// TwinCAT 3 PLC project MAIN
// ProgramVersion: 3.1.0.5
// libraries:
//   Tc2_ModbusRTU, * (Beckhoff Automation GmbH)
//   Tc2_Standard, * (Beckhoff Automation GmbH)
//   Tc2_System, * (Beckhoff Automation GmbH)
//   Tc2_Utilities, * (Beckhoff Automation GmbH)
//   Tc2_XmlDataSrv, * (Beckhoff Automation GmbH)
//   Tc3_Interfaces, * (Beckhoff Automation GmbH)
//   Tc3_Module, * (Beckhoff Automation GmbH)
//   VisuDialogs, * (System)
// project tree:
//   DUTs/ RESET_STATE.TcDUT, ST_DisplayPositions.TcDUT, ST_SavedStructure.TcDUT, ST_SavedPositions.TcDUT, SYSTEM_STATE.TcDUT
//   / GlobalTextList.TcGTLO, PlcTask.TcTTO, Visualization Manager.TcVMO (not stored), VISU_TASK.TcTTO
//   GVLs/ GV_HMI.TcGVL, GV_LIFT.TcGVL, GV_MODBUS.TcGVL
//   POUs/ HMI.TcPOU, IO_SWITCHBOARD.TcPOU, MAIN.TcPOU, MOVE_TO_POSITION.TcPOU, SYSTEM_RESET.TcPOU, XML.TcPOU
//   POUs/HMI/ HMI_Crush_Indicator.TcPOU, HMI_Door_Toggle.TcPOU, HMI_Down_Arrow_Indicator.TcPOU, HMI_Hard_Limits.TcPOU, HMI_System_Indicator.TcPOU, HMI_Ultimate_Limit.TcPOU, HMI_Up_Arrow_Indicator.TcPOU
//   POUs/Pendant Screen/ DoorFaults.TcPOU, DownLimit.TcPOU, EStop.TcPOU, JogLift.TcPOU, MoveToPosition.TcPOU, ReadWriteScreen.TcPOU, SelectSpike.TcPOU, SwitchScreens.TcPOU, UpLimit.TcPOU
//   POUs/Pendant Screen/Functions/ Execute_Write_Screen.TcPOU, Fill_Row_Four.TcPOU, Fill_Row_Three.TcPOU, Fill_Row_Two.TcPOU, Get_Valid_Indexs.TcPOU, Position_To_Row_Array.TcPOU, Spike_To_Half_Row_Array.TcPOU, Spike_To_Row_Array.TcPOU
//   VISUs/ MAIN_DASHBOARD.TcVIS, SAFETY_PANEL.TcVIS, TARGET_PANEL.TcVIS
// real-time tasks:
//   TASK PlcTask: cycle T#15ms, priority 20, ADS port 350
//   TASK VISU_TASK: cycle T#20ms, priority 30, ADS port 351
// I/O:
//   DEVICE Device 1 (EtherCAT), AmsNetId 5.31.29.63.2.1
//     Term 1 (EK1200) [EK1200-5000 EtherCAT Power supply (2A E-Bus)]
//       Term 2 (EL1904) [EL1904, 4 Ch. Safety Input 24V, TwinSAFE]
//         modules: Module 1 (FSOES)
//       Term 3 (EL1859) [EL1859 8Ch. Dig. Input 24V, 3ms, 8Ch. Dig. Output 24V, 0.5A]
//       Term 4 (EK1110) [EK1110 EtherCAT extension]
//     Term 5 (EK1914) [EK1914, 2 Ch. Safety Input/Output 24V,  TwinSAFE]
//       modules: Module 1 (FSOE), Module 2 (DIO)
//       Term 6 (EL1904) [EL1904, 4 Ch. Safety Input 24V, TwinSAFE]
//         modules: Module 1 (FSOES)
//       Term 7 (EL6021) [EL6021 Interface (RS422/485)]
//       Term 15 (EL9011) [EL9011 End Terminal]
//     Term 8 (EK1100) [EK1100 EtherCAT Coupler (2A E-Bus)]
//       Term 9 (EL6900) [EL6900, TwinSAFE PLC]
//       Term 10 (EL1904) [EL1904, 4 Ch. Safety Input 24V, TwinSAFE]
//         modules: Module 1 (FSOES)
//       Term 11 (EL1904) [EL1904, 4 Ch. Safety Input 24V, TwinSAFE]
//         modules: Module 1 (FSOES)
//       Term 12 (EL1904) [EL1904, 4 Ch. Safety Input 24V, TwinSAFE]
//         modules: Module 1 (FSOES)
//       Term 13 (EL1904) [EL1904, 4 Ch. Safety Input 24V, TwinSAFE]
//         modules: Module 1 (FSOES)
//       Term 16 (EL9011) [EL9011 End Terminal]
//     Box 14 (SICK AFS60A ST, 18-Bit) [AFS60A_ST 18-Bit]
// variable links:
//   Device 1 (EtherCAT) <-> Device 1 (EtherCAT)/Term 1 (EK1200)/Term 2 (EL1904)
//     Term 8 (EK1100)/ConnectionOutputs/Message_86 RxPDO <-> Module 1 (FSOES)/TxPDO/FSOE
//     Term 8 (EK1100)/Term 9 (EL6900)/ConnectionOutputs/Message_86 RxPDO <-> Module 1 (FSOES)/TxPDO/FSOE
//   Device 1 (EtherCAT) <-> Device 1 (EtherCAT)/Term 5 (EK1914)
//     Term 8 (EK1100)/Term 9 (EL6900)/ConnectionInputs/Message_87 TxPDO <-> Module 1 (FSOE)/Outputs/FSOE
//   Device 1 (EtherCAT) <-> Device 1 (EtherCAT)/Term 5 (EK1914)/Term 6 (EL1904)
//     Term 8 (EK1100)/Term 9 (EL6900)/ConnectionOutputs/Message_88 RxPDO <-> Module 1 (FSOES)/TxPDO/FSOE
//   Device 1 (EtherCAT) <-> Device 1 (EtherCAT)/Term 8 (EK1100)
//     Term 5 (EK1914)/Term 6 (EL1904)/Module 1 (FSOES)/TxPDO/FSOE <-> ConnectionOutputs/Message_88 RxPDO
//     Term 8 (EK1100)/Term 11 (EL1904)/Module 1 (FSOES)/TxPDO/FSOE <-> ConnectionOutputs/Message_90 RxPDO
//     Term 8 (EK1100)/Term 13 (EL1904)/Module 1 (FSOES)/TxPDO/FSOE <-> ConnectionOutputs/Message_92 RxPDO
//   Device 1 (EtherCAT) <-> Device 1 (EtherCAT)/Term 8 (EK1100)/Term 10 (EL1904)
//     Term 8 (EK1100)/ConnectionOutputs/Message_89 RxPDO <-> Module 1 (FSOES)/TxPDO/FSOE
//     Term 8 (EK1100)/Term 9 (EL6900)/ConnectionInputs/Message_89 TxPDO <-> Module 1 (FSOES)/RxPDO/FSOE
//   Device 1 (EtherCAT) <-> Device 1 (EtherCAT)/Term 8 (EK1100)/Term 11 (EL1904)
//     Term 8 (EK1100)/Term 9 (EL6900)/ConnectionOutputs/Message_90 RxPDO <-> Module 1 (FSOES)/TxPDO/FSOE
//   Device 1 (EtherCAT) <-> Device 1 (EtherCAT)/Term 8 (EK1100)/Term 12 (EL1904)
//     Term 8 (EK1100)/ConnectionOutputs/Message_91 RxPDO <-> Module 1 (FSOES)/TxPDO/FSOE
//     Term 8 (EK1100)/Term 9 (EL6900)/ConnectionInputs/Message_91 TxPDO <-> Module 1 (FSOES)/RxPDO/FSOE
//   Device 1 (EtherCAT) <-> Device 1 (EtherCAT)/Term 8 (EK1100)/Term 13 (EL1904)
//     Term 8 (EK1100)/Term 9 (EL6900)/ConnectionOutputs/Message_92 RxPDO <-> Module 1 (FSOES)/TxPDO/FSOE
//   Device 1 (EtherCAT) <-> Device 1 (EtherCAT)/Term 8 (EK1100)/Term 9 (EL6900)
//     Term 1 (EK1200)/Term 2 (EL1904)/Module 1 (FSOES)/RxPDO/FSOE <-> ConnectionInputs/Message_86 TxPDO
//     Term 5 (EK1914)/Term 6 (EL1904)/Module 1 (FSOES)/RxPDO/FSOE <-> ConnectionInputs/Message_88 TxPDO
//     Term 8 (EK1100)/Term 11 (EL1904)/Module 1 (FSOES)/RxPDO/FSOE <-> ConnectionInputs/Message_90 TxPDO
//     Term 8 (EK1100)/Term 13 (EL1904)/Module 1 (FSOES)/RxPDO/FSOE <-> ConnectionInputs/Message_92 TxPDO
//     Term 5 (EK1914)/Module 1 (FSOE)/Inputs/FSOE <-> ConnectionOutputs/Message_87 RxPDO
//     Term 8 (EK1100)/Term 10 (EL1904)/Module 1 (FSOES)/TxPDO/FSOE <-> ConnectionOutputs/Message_89 RxPDO
//     Term 8 (EK1100)/Term 12 (EL1904)/Module 1 (FSOES)/TxPDO/FSOE <-> ConnectionOutputs/Message_91 RxPDO
//   MAIN/MAIN Instance <-> Device 1 (EtherCAT)/Box 14 (SICK AFS60A ST, 18-Bit)
//     PlcTask Inputs/MOVE_TO_POSITION.currentRawPosition <-> TxPDO-1/Position Value
//   MAIN/MAIN Instance <-> Device 1 (EtherCAT)/Term 1 (EK1200)/Term 3 (EL1859)
//     PlcTask Inputs/GV_LIFT.LIMIT_OVERRIDE_BUTTON_IN <-> Channel 1/Input
//     PlcTask Inputs/IO_SWITCHBOARD.CONSOLE_DOWN_BUTTON_IN <-> Channel 3/Input
//     PlcTask Inputs/IO_SWITCHBOARD.CONSOLE_RESET_BUTTON_IN <-> Channel 5/Input
//     PlcTask Inputs/IO_SWITCHBOARD.CONSOLE_RUN_BUTTON_IN <-> Channel 4/Input
//     PlcTask Inputs/IO_SWITCHBOARD.CONSOLE_UP_BUTTON_IN <-> Channel 2/Input
//   MAIN/MAIN Instance <-> Device 1 (EtherCAT)/Term 5 (EK1914)
//     PlcTask Inputs/IO_SWITCHBOARD.REMOTE_DOWN_BUTTON_IN <-> Module 2 (DIO)/DIO Inputs/Input 1
//     PlcTask Inputs/IO_SWITCHBOARD.REMOTE_RESET_BUTTON_IN <-> Module 2 (DIO)/DIO Inputs/Input 0
//     PlcTask Inputs/IO_SWITCHBOARD.REMOTE_RUN_BUTTON_IN <-> Module 2 (DIO)/DIO Inputs/Input 3
//     PlcTask Inputs/IO_SWITCHBOARD.REMOTE_UP_BUTTON_IN <-> Module 2 (DIO)/DIO Inputs/Input 2
//   MAIN/MAIN Instance <-> Device 1 (EtherCAT)/Term 5 (EK1914)/Term 7 (EL6021)
//     PlcTask Inputs/GV_MODBUS.screen.InData/D[{0..21}] <-> COM TxPDO-Map Inputs/Data In {0..21}  (22 links)
//     PlcTask Inputs/GV_MODBUS.screen.InData/Status <-> COM TxPDO-Map Inputs/Status
//     PlcTask Outputs/GV_MODBUS.screen.OutData/Ctrl <-> COM RxPDO-Map Outputs/Ctrl
//     PlcTask Outputs/GV_MODBUS.screen.OutData/D[{0..21}] <-> COM RxPDO-Map Outputs/Data Out {0..21}  (22 links)
//   MAIN/MAIN Instance <-> Device 1 (EtherCAT)/Term 8 (EK1100)/Term 9 (EL6900)
//     PlcTask Inputs/GV_LIFT.CONSOLE_ESTOP_INDICATOR_IN <-> StandardInputs/Standard Out Var 68
//     PlcTask Inputs/GV_LIFT.CRUSH_PROTECTION_INDICATOR_IN <-> StandardInputs/Standard Out Var 60
//     PlcTask Inputs/GV_LIFT.DOOR_{1..4}_INDICATOR_IN <-> StandardInputs/Standard Out Var {56..59}  (4 links)
//     PlcTask Inputs/GV_LIFT.DOOR_{1..4}_INDICATOR_LATCH_IN <-> StandardInputs/Standard Out Var {72..75}  (4 links)
//     PlcTask Inputs/GV_LIFT.DOWNSTAGE_ESTOP_INDICATOR_IN <-> StandardInputs/Standard Out Var 70
//     PlcTask Inputs/GV_LIFT.DOWN_INDICATOR_IN <-> StandardInputs/Standard Out Var 63
//     PlcTask Inputs/GV_LIFT.DOWN_LIMIT_INDICATOR_IN <-> StandardInputs/Standard Out Var 65
//     PlcTask Inputs/GV_LIFT.DOWN_LIMIT_INDICATOR_LATCH_IN <-> StandardInputs/Standard Out Var 77
//     PlcTask Inputs/GV_LIFT.ESTOP_INDICATOR_IN <-> StandardInputs/Standard Out Var 61
//     PlcTask Inputs/GV_LIFT.FAULT_INDICATOR_IN <-> StandardInputs/Standard Out Var 62
//     PlcTask Inputs/GV_LIFT.PIT_ESTOP_INDICATOR_IN <-> StandardInputs/Standard Out Var 67
//     PlcTask Inputs/GV_LIFT.PUMP_ESTOP_INDICATOR_IN <-> StandardInputs/Standard Out Var 69
//     PlcTask Inputs/GV_LIFT.REMOTE_ESTOP_INDICATOR_IN <-> StandardInputs/Standard Out Var 71
//     PlcTask Inputs/GV_LIFT.ULTIMATE_LIMIT_INDICATOR_IN <-> StandardInputs/Standard Out Var 66
//     PlcTask Inputs/GV_LIFT.ULTIMATE_LIMIT_INDICATOR_LATCH_IN <-> StandardInputs/Standard Out Var 78
//     PlcTask Inputs/GV_LIFT.UPSTAGE_ESTOP_INDICATOR_IN <-> StandardInputs/Standard Out Var 55
//     PlcTask Inputs/GV_LIFT.UP_INDICATOR_IN <-> StandardInputs/Standard Out Var 54
//     PlcTask Inputs/GV_LIFT.UP_LIMIT_INDICATOR_IN <-> StandardInputs/Standard Out Var 64
//     PlcTask Inputs/GV_LIFT.UP_LIMIT_INDICATOR_LATCH_IN <-> StandardInputs/Standard Out Var 76
//     PlcTask Outputs/GV_LIFT.DOWN_BUTTON_OUT <-> StandardOutputs/Standard In Var 53
//     PlcTask Outputs/GV_LIFT.UP_BUTTON_OUT <-> StandardOutputs/Standard In Var 52
//     PlcTask Outputs/SYSTEM_RESET.ERROR_ACKNOWLEDGEMENT_BUTTON_OUT <-> StandardOutputs/Standard In Var 1
//     PlcTask Outputs/SYSTEM_RESET.ESTOP_RESTART_BUTTON_OUT <-> StandardOutputs/Standard In Var 10

CONFIGURATION MAIN
    RESOURCE PLC ON TwinCAT3
        TASK PlcTask(INTERVAL := T#20ms, PRIORITY := 20);
        TASK VISU_TASK(INTERVAL := T#30ms, PRIORITY := 30);
        PROGRAM MAIN WITH PlcTask : MAIN;
        PROGRAM VisuElems_Visu_Prg WITH VISU_TASK : VisuElems.Visu_Prg;
    END_RESOURCE
END_CONFIGURATION

// ---- DUTs/RESET_STATE.TcDUT
{attribute 'qualified_only'}
{attribute 'strict'}
TYPE RESET_STATE :
(
	IDLE,
	ERRACK_ON,
	ERRACK_OFF,
	IDLE2,
	ESTOP_RESET_ON,
	COMPLETE
);
END_TYPE

// ---- DUTs/ST_DisplayPositions.TcDUT
TYPE ST_DisplayPositions :
STRUCT
	target		:	STRING;
	description	:	STRING;
END_STRUCT
END_TYPE

// ---- DUTs/ST_SavedStructure.TcDUT
TYPE ST_SavedStructure :
STRUCT
	rStagePosition 	:	REAL;
	UpSoftLim		:	REAL;
	DownSoftLim		:	REAL;
	Counter			:	INT;
	SavedPos		:	ARRAY [1..25] OF ST_SavedPositions;
END_STRUCT
END_TYPE

// ---- DUTs/ST_SavedPositions.TcDUT
TYPE ST_SavedPositions :
STRUCT
	target		:	REAL;
	description	:	STRING;
	targetclear	:	BOOL:=FALSE;
END_STRUCT
END_TYPE

// ---- DUTs/SYSTEM_STATE.TcDUT
{attribute 'qualified_only'}
{attribute 'strict'}
TYPE SYSTEM_STATE :
(
	SYSTEM_READY,
	CONSOLE_CONTROL,
	REMOTE_CONTROL
);
END_TYPE

// ---- GVLs/GV_HMI.TcGVL
{attribute 'qualified_only'}
VAR_GLOBAL CONSTANT
	iMaxTargets		:	INT:=25;
	iMaxButtons		:	INT:=20;

END_VAR

VAR_GLOBAL
	ColorToggle		  :	ARRAY [1..20] OF BOOL;

	CurrentPos		:	REAL:=100;
	updatedPos  	:   REAL;
	RowSelect		:	INT:=1;
	ColumnSelect	:	INT:=1;
	RowSelected		:	INT:= RowSelect;


	dwRed				: DWORD:= 16#FFFF0000;
	dwGreen				: DWORD:= 16#FF008040;
	dwYellow			: DWORD:= 16#FFFFFF00;
	dwGrey				: DWORD:= 16#FFBEBEBE;
	
END_VAR

// ---- GVLs/GV_LIFT.TcGVL
{attribute 'qualified_only'}

(*
Signal Flow:

 Physical/HMI Button ---> *_BUTTON_IN ---> *_BUTTON_OUT ---> *_SAFETY_IN ---> *_SAFETY_OUT ---> *_INDICATOR_IN ---> *_INDICATOR_OUT
|------PHYSICAL-----|    |--------IO_SWITCHBOARD-------|    |-------SAFETY PROJECT--------|    |-----------IO_SWITCHBOARD-----------|

This convolution is based on the alias device scheme in the safety project. Recall that an input alias in the safety project must be 
mapped to a PLC/Physical output, and vice versa. The IO_SWITCHBOARD handles signal passthroughs and negotiations between operator
stations. Variables in this GVL should reflect the accurate state of signals to/from the machine. As such, the UP/DOWN/RUN buttons
should reference the appropriate local variables in IO_SWITCHBOARD, which will route signals to the UP/DOWN/RUN_BUTTON_OUT outputs in
this GVL.
*)
VAR_GLOBAL
	REMOTE_ACTIVE_INDICATOR_OUT AT %Q* : BOOL;
	CONSOLE_ACTIVE_INDICATOR_OUT AT %Q* : BOOL;
	
	SYSTEM_RESET_BUTTON_IN AT %I*: BOOL;
	
	//UP_BUTTON_IN AT %I* : BOOL;
	UP_BUTTON_OUT AT %Q* : BOOL;
	
	UP_INDICATOR_IN AT %I* : BOOL;
	UP_INDICATOR_OUT AT %Q* : BOOL;
	
	//DOWN_BUTTON_IN AT %I* : BOOL;
	DOWN_BUTTON_OUT AT %Q* : BOOL;
	
	DOWN_INDICATOR_IN AT %I* : BOOL;
	DOWN_INDICATOR_OUT AT %Q* : BOOL;

	//RUN_BUTTON_IN AT %I* : BOOL;
	RUN_BUTTON_OUT AT %Q* : BOOL;
	
	DOOR_1_INDICATOR_IN AT %I* : BOOL;
	DOOR_1_INDICATOR_OUT AT %Q* : BOOL;
	
	DOOR_1_INDICATOR_LATCH_IN AT %I* : BOOL;
	DOOR_1_INDICATOR_LATCH_OUT AT %Q* : BOOL;
	
	DOOR_2_INDICATOR_IN AT %I* : BOOL;
	DOOR_2_INDICATOR_OUT AT %Q* : BOOL;
	
	DOOR_2_INDICATOR_LATCH_IN AT %I* : BOOL;
	DOOR_2_INDICATOR_LATCH_OUT AT %Q* : BOOL;
	
	DOOR_3_INDICATOR_IN AT %I* : BOOL;
	DOOR_3_INDICATOR_OUT AT %Q* : BOOL;
	
	DOOR_3_INDICATOR_LATCH_IN AT %I* : BOOL;
	DOOR_3_INDICATOR_LATCH_OUT AT %Q* : BOOL;
	
	DOOR_4_INDICATOR_IN AT %I* : BOOL;
	DOOR_4_INDICATOR_OUT AT %Q* : BOOL;
	
	DOOR_4_INDICATOR_LATCH_IN AT %I* : BOOL;
	DOOR_4_INDICATOR_LATCH_OUT AT %Q* : BOOL;
	
	DOWN_LIMIT_INDICATOR_IN AT %I* : BOOL;
	DOWN_LIMIT_INDICATOR_OUT AT %Q* : BOOL;
	
	DOWN_LIMIT_INDICATOR_LATCH_IN AT %I* : BOOL;
	DOWN_LIMIT_INDICATOR_LATCH_OUT AT %Q* : BOOL;
	
	UP_LIMIT_INDICATOR_IN AT %I* : BOOL;
	UP_LIMIT_INDICATOR_OUT AT %Q* : BOOL;
	
	UP_LIMIT_INDICATOR_LATCH_IN AT %I* : BOOL;
	UP_LIMIT_INDICATOR_LATCH_OUT AT %Q* : BOOL;
	
	ULTIMATE_LIMIT_INDICATOR_IN AT %I* : BOOL;
	ULTIMATE_LIMIT_INDICATOR_OUT AT %Q* : BOOL;
	
	ULTIMATE_LIMIT_INDICATOR_LATCH_IN AT %I* : BOOL;
	ULTIMATE_LIMIT_INDICATOR_LATCH_OUT AT %Q* : BOOL;
	
	CRUSH_PROTECTION_INDICATOR_IN AT %I* : BOOL;
	CRUSH_PROTECTION_INDICATOR_OUT AT %Q* : BOOL;
	
	FAULT_INDICATOR_IN AT %I* : BOOL;
	FAULT_INDICATOR_OUT AT %Q* : BOOL;
	
	ESTOP_INDICATOR_IN AT %I* : BOOL;
	ESTOP_INDICATOR_OUT AT %Q* : BOOL;
	
	REMOTE_ESTOP_INDICATOR_IN AT %I* : BOOL;
	REMOTE_ESTOP_INDICATOR_OUT AT %Q* : BOOL;
	
	PIT_ESTOP_INDICATOR_IN AT %I* : BOOL;
	PIT_ESTOP_INDICATOR_OUT AT %Q* : BOOL;
	
	PUMP_ESTOP_INDICATOR_IN AT %I* : BOOL;
	PUMP_ESTOP_INDICATOR_OUT AT %Q* : BOOL;
	
	DOWNSTAGE_ESTOP_INDICATOR_IN AT %I* : BOOL;
	DOWNSTAGE_ESTOP_INDICATOR_OUT AT %Q* : BOOL;
	
	UPSTAGE_ESTOP_INDICATOR_IN AT %I* : BOOL;
	UPSTAGE_ESTOP_INDICATOR_OUT AT %Q* : BOOL;
	
	CONSOLE_ESTOP_INDICATOR_IN AT %I* : BOOL;
	CONSOLE_ESTOP_INDICATOR_OUT AT %Q* : BOOL;
	
	TARGET_POSITION : REAL;
	CURRENT_POSITION : REAL;
	
	MTP_ALLOWED : BOOL := FALSE;
	JUST_RAN: BOOL := FALSE;
	
	SYSTEM_FAULT : BOOL;
	
	LIMIT_OVERRIDE_BUTTON_IN AT %I* : BOOL;
	
	STAGE_POSITION : REAL;
END_VAR

// ---- GVLs/GV_MODBUS.TcGVL
{attribute 'qualified_only'}
VAR_GLOBAL CONSTANT
	UnitID: BYTE := 101;	
	timeout: TIME := T#1S;
	quantity: WORD := 5;
	
	btnUp: WORD := 2;
	btnDwn: WORD := 4;
	btnEnter: WORD := 1;
	
	oneLeftAddr: WORD := 0;
	oneRightAddr: WORD:= 5;
	twoLeftAddr: WORD:= 10;
	twoRightAddr: WORD:= 15;
	threeLeftAddr: WORD:= 20;
	threeRightAddr: WORD:= 25;
	fourLeftAddr: WORD:= 30;
	fourRightAddr: WORD:= 35;	
	
	blank: ARRAY [1..5] OF WORD := [16#2020, 16#2020, 16#2020, 16#2020, 16#2020];
	ok: ARRAY [1..5] OF WORD := [16#4F4B, 16#2020, 16#2020, 16#2020, 16#2020];
	fault_string: ARRAY [1..5] OF WORD := [16#4641, 16#554C, 16#5420, 16#2020, 16#2020];
	engaged : ARRAY [1..5] OF WORD := [16#454E, 16#4741, 16#4745, 16#4420, 16#2020];

	inch: WORD:= 16#22;
	inchSpace: WORD:= 16#2220;
	space: WORD:= 16#0020;
	spaceASCII: STRING := ' ';
	dblSpace: WORD:=16#2020;
	selected: WORD:= 16#3E;
	selectedASCII: STRING:= '>';
	loaded: WORD:= 16#2A;
	loadedASCII: STRING:= '*';
	outOfBoundsASCII: STRING := 'x';
	
	filterTarget: REAL:= 999.99;
END_VAR

VAR_GLOBAL	
	
	screen: ModbusRtuMasterV2_KL6x22B;
	writeExecute: BOOL := TRUE;
	readExecute: BOOL := FALSE;
	doneWriting: BOOL := FALSE;
	
	oneLeft: ARRAY [1..5] OF WORD := GV_MODBUS.blank;
	oneRight: ARRAY [1..5] OF WORD;                              
	twoLeft: ARRAY [1..5] OF WORD;
	twoRight: ARRAY [1..5] OF WORD;	                               
	threeLeft: ARRAY [1..5] OF WORD;
	threeRight: ARRAY [1..5] OF WORD;	                               
	fourLeft: ARRAY [1..5] OF WORD; 
	fourRight: ARRAY [1..5] OF WORD;
				
	addr: WORD:= GV_MODBUS.oneLeftAddr;
	data: ARRAY [1..5] OF WORD := GV_MODBUS.oneLeft;	
	
	btnData: WORD := 0;		
	
	wasMTS : BOOL := FALSE;
	refreshInterval: INT := 50;
END_VAR

// ---- POUs/MAIN.TcPOU
PROGRAM MAIN
VAR		

END_VAR

IF GV_LIFT.DOOR_1_INDICATOR_LATCH_IN THEN
	GV_LIFT.DOOR_1_INDICATOR_LATCH_OUT := TRUE;
ELSE
	GV_LIFT.DOOR_1_INDICATOR_LATCH_OUT := FALSE;	
END_IF

IF GV_LIFT.PIT_ESTOP_INDICATOR_IN THEN
	GV_LIFT.PIT_ESTOP_INDICATOR_OUT := TRUE;
ELSE
	GV_LIFT.PIT_ESTOP_INDICATOR_OUT := FALSE;	
END_IF

IF GV_LIFT.DOWNSTAGE_ESTOP_INDICATOR_IN THEN
	GV_LIFT.DOWNSTAGE_ESTOP_INDICATOR_OUT := TRUE;
ELSE
	GV_LIFT.DOWNSTAGE_ESTOP_INDICATOR_OUT := FALSE;	
END_IF

IF GV_LIFT.ESTOP_INDICATOR_IN THEN
	GV_LIFT.ESTOP_INDICATOR_OUT := TRUE;
ELSE
	GV_LIFT.ESTOP_INDICATOR_OUT := FALSE;	
END_IF

IF GV_LIFT.FAULT_INDICATOR_IN THEN
	GV_LIFT.FAULT_INDICATOR_OUT := TRUE;
ELSE
	GV_LIFT.FAULT_INDICATOR_OUT := FALSE;	
END_IF

IF GV_LIFT.UP_BUTTON_IN THEN
	GV_LIFT.UP_BUTTON_OUT := TRUE;
ELSE
	GV_LIFT.UP_BUTTON_OUT := FALSE;
END_IF

IF GV_LIFT.DOWN_BUTTON_IN THEN
	GV_LIFT.DOWN_BUTTON_OUT := TRUE;
ELSE
	GV_LIFT.DOWN_BUTTON_OUT := FALSE;
END_IF

IF GV_LIFT.RUN_BUTTON_IN THEN
	GV_LIFT.RUN_BUTTON_OUT := TRUE;
ELSE
	GV_LIFT.RUN_BUTTON_OUT := FALSE;
END_IF

XML(); 
//HMI();
IO_SWITCHBOARD();
SYSTEM_RESET();
MOVE_TO_POSITION();
SwitchScreens();

END_PROGRAM

// ---- POUs/XML.TcPOU
 PROGRAM XML
VAR
   savedvalues     : ST_SavedStructure;
   fbXmlSrvWrite   : FB_XmlSrvWrite;
   fbXmlSrvRead    : FB_XmlSrvRead; 
   sFileFolder     : T_MaxString := '\Hard Disk\'; (* CE: '\Hard Disk\' *) (* Win10: '\C:\ *)
   sFileName       : T_MaxString := 'HMI-Saved-Positions.xml';
   //sFilePath 	   : T_MaxString := 'C:\HMI-Saved-Positions.xml';  				//disable for CE
   sFilePath       : T_MaxString := '\Hard Disk\HMI-Saved-Positions.xml';		//enable for CE
   (*sFilePathWrite = sFileFolder + time + sFileName*)
   bExecute        : BOOL; 
   sXPath          : T_MaxString := '/dataentry/MAIN.savedvalues';
   ntGetTime       : NT_GetTime;
   stMyTimestruct  : TIMESTRUCT;
   iState          : INT := 0;
   bTwentySec      : BOOL:= FALSE;
   bButton         : BOOL:= FALSE;
   bTwentySecOver  : BOOL;
   triggerWrite    : R_TRIG;
   triggerButton   : R_TRIG;
   i			   : INT:=1;
   LoadComplate   : BOOL;
END_VAR

triggerButton(CLK:= bButton);


CASE iState OF
0: (* initialize *)
   fbXmlSrvRead(
   	 pSymAddr  := ADR(savedvalues),
     cbSymSize := SIZEOF(savedvalues), 
     sFilePath := sFilePath,
     sXPath    := sXPath,
     bExecute  := TRUE
   );
   iState:= 1; 
   ;
   
1: (* wait for read operation *)
   fbXmlSrvRead(bExecute:= FALSE);
   IF NOT fbXmlSrvRead.bBusy AND NOT fbXmlSrvRead.bError THEN
     iState:= 2; 
	 LoadComplate := TRUE;
   ELSIF fbXmlSrvRead.bError THEN
     iState:= 100;
	 LoadComplate:=FALSE;
   END_IF
 
2: (* Write *)
	savedvalues.counter:=savedvalues.counter + 1;
	IF savedvalues.counter = 326767 THEN
		savedvalues.counter := 0;
	END_IF

   fbXmlSrvWrite(nMode:=XMLSRV_ADDMISSING, pSymAddr:= ADR(savedvalues),
   cbSymSize:= SIZEOF(savedvalues));
   ntGetTime(START:= TRUE, TIMESTR=>stMyTimestruct); (* get Windows time *)
   IF NOT ntGetTime.BUSY AND NOT ntGetTime.ERR THEN
      iState:= 5;
   ELSIF ntGetTime.ERR THEN
      iState:= 100;
 END_IF
   
5: (* working state *)
   ntGetTime(START:= FALSE);
   IF NOT ntGetTime.BUSY AND NOT ntGetTime.ERR THEN
      ntGetTime(START:= TRUE, TIMESTR=>stMyTimestruct);
   ELSIF ntGetTime.ERR THEN
      iState:= 100;
   END_IF

	IF (stMyTimestruct.wMinute = 0 AND stMyTimeStruct.wSecond = 5) OR (stMyTimestruct.wMinute = 15 AND stMyTimeStruct.wSecond = 5) OR (stMyTimeStruct.wMinute = 30 AND stMyTimeStruct.wSecond = 5) OR (stMyTimeStruct.wMinute = 45 AND stMyTimeStruct.wSecond = 5) OR (stMyTimeStruct.wMinute = 60 AND stMyTimeStruct.wSecond = 5) THEN
		bTwentySecOver:= TRUE;
		IF	GV_LIFT.STAGE_POSITION <> 0 THEN
			savedvalues.rStagePosition := GV_LIFT.STAGE_POSITION;
		END_IF
	ELSE
		bTwentySecOver:= FALSE;
	END_IF
	
   (* if 20s have passed => trigger writing-process *)
   triggerWrite(CLK:=bTwentySecOver);
   IF (triggerWrite.Q OR triggerButton.Q) AND NOT fbXmlSrvWrite.bBusy AND NOT fbXmlSrvWrite.bError THEN 
      (* write *)
      fbXmlSrvWrite(sFilePath:=sFilePath, sXPath:=sXPath, bExecute:= TRUE);

   ELSIF fbXmlSrvWrite.bError THEN
      iState:= 100;
   END_IF

   (* reset fbXmlSrvWrite *)
   IF fbXmlSrvWrite.bBusy AND NOT ntGetTime.ERR THEN
      fbXmlSrvWrite(bExecute:= FALSE);
   ELSIF ntGetTime.ERR THEN
      iState:= 100;
   END_IF
 
100: (* error state*) 
 ;

END_CASE

END_PROGRAM

// ---- POUs/HMI.TcPOU
PROGRAM HMI
VAR
	displayvalues		: ARRAY[1..25] OF ST_DisplayPositions;
	displaycounter		: INT:=1;
	insidelimits		: BOOL:= FALSE;
	bLoadOK				: BOOL:= FALSE;
	bLoaded				: BOOL:= FALSE;
	bUnload				: BOOL:= FALSE;
	bTgtLoaded			: BOOL:= FALSE;
	bEditEnable			: BOOL:= FALSE;
	DisplayTgtPos	:	STRING:= '';	
	
//Indicator Flags	
	bSoftUpLimFlag		: BOOL;
	bSoftDownLimFlag	: BOOL;
	bSoftLimFlag		: BOOL;
	bLimitHeaderFlag	: BOOL;
	bSystemFlag			: BOOL:= FALSE;
		
//Color Fields
	dwUpArrow			: DWORD;
	dwDownArrow			: DWORD;
	dwDoorFlag			: DWORD;
	dwDoor1				: DWORD;
	dwDoor2				: DWORD;
	dwDoor3				: DWORD;
	dwDoor4				: DWORD;
	dwCrushFlag			: DWORD;
	dwSysFaultFlag		: DWORD;

END_VAR

//Displayed Values Logic
	CASE displaycounter OF
	1..25: (* Creates a state machine that will write XML values to displayed values *)
		IF 	XML.savedvalues.SavedPos[displaycounter].targetclear = FALSE THEN 
			displayvalues[displaycounter].target := '';
			//displayvalues[displaycounter].description := '';
		ELSE	
			displayvalues[displaycounter].target := CONCAT((REAL_TO_STRING(XML.savedvalues.SavedPos[displaycounter].target)),'"');
		END_IF
		displaycounter := displaycounter +1;
	26: (*Resets State Machine *)
			displaycounter := 1;
	END_CASE
	
	displayvalues[displaycounter].description := (XML.savedvalues.SavedPos[displaycounter].description);	
	
//Determines if Target is inside Soft Limits
	IF XML.savedvalues.savedpos[GV_HMI.RowSelect].target <= (XML.savedvalues.UpSoftLim) AND XML.savedvalues.savedpos[GV_HMI.RowSelect].target >= (XML.savedvalues.DownSoftLim) THEN
		insidelimits := TRUE;
	ELSE
		insidelimits := FALSE;
	END_IF
	
//Load Button Logic
	IF XML.savedvalues.savedpos[GV_HMI.RowSelect].targetclear AND insidelimits AND NOT GV_LIFT.RUN_BUTTON_OUT THEN
		bLoadOK	:= TRUE;
	ELSE
		bLoadOK	:= FALSE;	
	END_IF

//Removing Target if highlighted target changes
	IF xml.savedvalues.SavedPos[GV_HMI.RowSelected].target <> xml.savedvalues.SavedPos[GV_HMI.RowSelect].target THEN
		bTgtLoaded := FALSE;
	END_IF
	
// Displaying Loaded Target
		DisplayTgtPos:= CONCAT(REAL_TO_STRING((GV_LIFT.TARGET_POSITION)),'"');

// Hiding load Button to Display Unload Button
	IF bLoadOK = TRUE AND bTgtLoaded = TRUE AND GV_LIFT.MTS_ALLOWED THEN
		bUnload := TRUE;
	ELSE bUnload := FALSE;	
	END_IF

//System Indicator

//Soft Up Limit Indicator
	IF (GV_LIFT.CURRENT_POSITION > XML.savedvalues.UpSoftLim) AND NOT GV_LIFT.LIMIT_OVERRIDE_BUTTON_IN THEN
		bSoftUpLimFlag := FALSE;
	ELSE bSoftUpLimFlag := TRUE;
	END_IF
	
//Soft Down Limit Indicator
	IF (GV_LIFT.CURRENT_POSITION < XML.savedvalues.DownSoftLim) AND NOT GV_LIFT.LIMIT_OVERRIDE_BUTTON_IN THEN
		bSoftDownLimFlag := FALSE;
	ELSE bSoftDownLimFlag := TRUE;
	END_IF
		
//Soft Limit System Indicator
	IF (GV_LIFT.CURRENT_POSITION < XML.savedvalues.DownSoftLim) OR (GV_LIFT.CURRENT_POSITION < XML.savedvalues.UpSoftLim) OR GV_LIFT.LIMIT_OVERRIDE_BUTTON_IN THEN
		bSoftLimFlag := TRUE;
		bSystemFlag:= TRUE;
	ELSE bSoftLimFlag := FALSE;
	END_IF
	
//Limit Safety Page Header
	IF NOT bSoftLimFlag OR NOT GV_LIFT.UP_LIMIT_INDICATOR_IN OR NOT GV_LIFT.DOWN_LIMIT_INDICATOR_IN OR NOT GV_LIFT.ULTIMATE_LIMIT_INDICATOR_IN THEN
		bLimitHeaderFlag := FALSE;
	ELSE bLimitHeaderFlag := TRUE;
	END_IF
 	

//Button and Inidcator Calls
	HMI_Up_Arrow_Indicator();
	HMI_Down_Arrow_Indicator();
	HMI_Door_Toggle();
	HMI_Crush_Indicator();
	HMI_System_Indicator();
	HMI_Hard_Limits();
	HMI_Ultimate_Limit();

END_PROGRAM

// ---- POUs/HMI/HMI_Up_Arrow_Indicator.TcPOU
PROGRAM HMI_Up_Arrow_Indicator
VAR
	dwUpArrow: DWORD;
END_VAR

IF NOT GV_LIFT.UP_LIMIT_INDICATOR_IN THEN 
	dwUpArrow := GV_HMI.dwRed;
ELSIF GV_LIFT.CURRENT_POSITION > XML.savedvalues.UpSoftLim THEN
	dwUpArrow := GV_HMI.dwYellow;
ELSIF GV_LIFT.UP_INDICATOR_IN THEN
	 dwUpArrow := GV_HMI.dwGreen;
ELSE
	dwUpArrow := GV_HMI.dwGrey;
END_IF

END_PROGRAM

// ---- POUs/HMI/HMI_Down_Arrow_Indicator.TcPOU
PROGRAM HMI_Down_Arrow_Indicator
VAR
	dwDownArrow: DWORD;
END_VAR

IF NOT GV_LIFT.DOWN_LIMIT_INDICATOR_IN THEN 
	dwDownArrow := GV_HMI.dwRed;
ELSIF GV_Lift.ULTIMATE_LIMIT_INDICATOR_OUT THEN
	dwDownArrow := GV_HMI.dwRed;
ELSIF GV_LIFT.CURRENT_POSITION < XML.savedvalues.DownSoftLim THEN
	dwDownArrow := GV_HMI.dwYellow;
ELSIF GV_LIFT.DOWN_INDICATOR_IN THEN
	 dwDownArrow := GV_HMI.dwGreen;
ELSE
	dwDownArrow := GV_HMI.dwGrey;
END_IF

END_PROGRAM

// ---- POUs/HMI/HMI_Door_Toggle.TcPOU
PROGRAM HMI_Door_Toggle
VAR
	dwDoorFlag: DWORD;
	dwDoor1: DWORD;
	dwDoor2: DWORD;
	dwDoor3: DWORD;
	dwDoor4: DWORD;
	bDoorFlag : BOOL;
END_VAR

//Door Interlock Indicator Logic
	IF GV_LIFT.DOOR_1_INDICATOR_IN AND GV_LIFT.DOOR_2_INDICATOR_IN AND GV_LIFT.DOOR_3_INDICATOR_IN AND GV_LIFT.DOOR_4_INDICATOR_IN THEN
		dwDoorFlag := GV_HMI.dwGreen;
		bDoorFlag := FALSE;
	ELSE dwDoorFlag := GV_HMI.dwRed;
		bDoorFlag := TRUE;
	END_IF 
	
	//Door 1 Indicator
		IF GV_LIFT.DOOR_1_INDICATOR_OUT THEN
			dwDoor1 := GV_HMI.dwRed;
		ELSIF GV_Lift.DOOR_1_INDICATOR_LATCH_OUT THEN
			dwDoor1 := GV_HMI.dwYellow;
		ELSE dwDoor1 := GV_HMI.dwGreen;
		END_IF
	//Door 2 Indicator
		IF GV_LIFT.DOOR_2_INDICATOR_OUT THEN
			dwDoor2 := GV_HMI.dwRed;
		ELSIF GV_Lift.DOOR_2_INDICATOR_LATCH_OUT THEN
			dwDoor2 := GV_HMI.dwYellow;
		ELSE dwDoor2 := GV_HMI.dwGreen;
		END_IF
	//Door 3 Indicator
		IF GV_LIFT.DOOR_3_INDICATOR_OUT THEN
			dwDoor3 := GV_HMI.dwRed;
		ELSIF GV_Lift.DOOR_3_INDICATOR_LATCH_OUT THEN
			dwDoor3 := GV_HMI.dwYellow;
		ELSE dwDoor3 := GV_HMI.dwGreen;
		END_IF
	//Door 4 Indicator
		IF GV_LIFT.DOOR_4_INDICATOR_OUT THEN
			dwDoor4 := GV_HMI.dwRed;
		ELSIF GV_Lift.DOOR_4_INDICATOR_LATCH_OUT THEN
			dwDoor4 := GV_HMI.dwYellow;
		ELSE dwDoor4 := GV_HMI.dwGreen;
		END_IF

END_PROGRAM

// ---- POUs/HMI/HMI_Crush_Indicator.TcPOU
PROGRAM HMI_Crush_Indicator
VAR
	dwCrushFlag: DWORD;
	bCrushFlag: BOOL;
END_VAR

IF GV_LIFT.CRUSH_PROTECTION_INDICATOR_IN THEN
	dwCrushFlag := GV_HMI.dwGreen;
	bCrushFlag := FALSE;
ELSE dwCrushFlag := GV_HMI.dwRed;
	bCrushFlag := TRUE;
END_IF

END_PROGRAM

// ---- POUs/HMI/HMI_System_Indicator.TcPOU
PROGRAM HMI_System_Indicator
VAR
	bSystemFlag : BOOL;
END_VAR

IF
	GV_LIFT.ESTOP_INDICATOR_OUT AND GV_LIFT.ULTIMATE_LIMIT_INDICATOR_IN AND GV_LIFT.UP_LIMIT_INDICATOR_IN AND GV_LIFT.DOWN_LIMIT_INDICATOR_IN AND HMI.bSoftLimFlag AND HMI_Door_Toggle.bDoorFlag = FALSE AND HMI_Crush_Indicator.bCrushFlag = FALSE THEN
	bSystemFlag := TRUE;
ELSE
	bSystemFlag := FALSE;
END_IF

END_PROGRAM

// ---- POUs/HMI/HMI_Hard_Limits.TcPOU
PROGRAM HMI_Hard_Limits
VAR
	UpHardLimit		: DWORD;
	DownHardLimit	: DWORD;
	HardLimitFlag	: DWORD;
END_VAR

IF GV_Lift.UP_LIMIT_INDICATOR_OUT THEN
	UpHardLimit := GV_HMI.dwRed;
ELSIF GV_Lift.UP_LIMIT_INDICATOR_LATCH_OUT THEN
	UpHardLimit := GV_HMI.dwYellow;
ELSE UpHardLimit := GV_HMI.dwGreen;
END_IF

IF GV_Lift.DOWN_LIMIT_INDICATOR_OUT THEN
	DownHardLimit := GV_HMI.dwRed;
ELSIF GV_Lift.DOWN_LIMIT_INDICATOR_LATCH_OUT THEN
	DownHardLimit := GV_HMI.dwYellow;
ELSE DownHardLimit := GV_HMI.dwGreen;
END_IF

IF GV_Lift.DOWN_LIMIT_INDICATOR_OUT OR GV_LIFT.UP_LIMIT_INDICATOR_OUT OR GV_LIFT.ULTIMATE_LIMIT_INDICATOR_OUT THEN
	HardLimitFlag := GV_HMI.dwRed;
ELSE HardLimitFlag := GV_HMI.dwGreen;
END_IF

END_PROGRAM

// ---- POUs/HMI/HMI_Ultimate_Limit.TcPOU
PROGRAM HMI_Ultimate_Limit
VAR
	DownUltLimit: DWORD;
END_VAR

IF GV_Lift.ULTIMATE_LIMIT_INDICATOR_OUT THEN
	DownUltLimit := GV_HMI.dwRed;
ELSIF GV_Lift.ULTIMATE_LIMIT_INDICATOR_LATCH_OUT THEN
	DownUltLimit := GV_HMI.dwYellow;
ELSE DownUltLimit := GV_HMI.dwGreen;
END_IF

END_PROGRAM

// ---- POUs/IO_SWITCHBOARD.TcPOU
PROGRAM IO_SWITCHBOARD
VAR CONSTANT
	STATE_TIMEOUT : INT := 50;
END_VAR
VAR
	state : SYSTEM_STATE;
	stateIdleCounter : INT;
	isConsoleActive : BOOL;
	isRemoteActive : BOOL;
	
	CONSOLE_DOWN_BUTTON_IN AT %I* : BOOL;
	CONSOLE_RUN_BUTTON_IN AT %I* : BOOL;
	CONSOLE_UP_BUTTON_IN AT %I* : BOOL;
	CONSOLE_RESET_BUTTON_IN AT %I* : BOOL;
	
END_VAR

isConsoleActive := (CONSOLE_DOWN_BUTTON_IN OR CONSOLE_RUN_BUTTON_IN OR CONSOLE_UP_BUTTON_IN);

CASE state OF 
	SYSTEM_STATE.SYSTEM_READY :
		GV_LIFT.CONSOLE_ACTIVE_INDICATOR_OUT := FALSE;
		GV_LIFT.REMOTE_ACTIVE_INDICATOR_OUT := FALSE;
		IF isConsoleActive THEN
			state := SYSTEM_STATE.CONSOLE_CONTROL;
		ELSIF isRemoteActive THEN
			state := SYSTEM_STATE.REMOTE_CONTROL;
		END_IF
		
	SYSTEM_STATE.CONSOLE_CONTROL :
		IF isConsoleActive THEN
			IF CONSOLE_RUN_BUTTON_IN THEN
				GV_LIFT.RUN_BUTTON_OUT := CONSOLE_RUN_BUTTON_IN;
			ELSE
				GV_LIFT.DOWN_BUTTON_OUT := (CONSOLE_DOWN_BUTTON_IN);
				GV_LIFT.UP_BUTTON_OUT := (CONSOLE_UP_BUTTON_IN);
			END_IF
			stateIdleCounter := 0;
			GV_LIFT.CONSOLE_ACTIVE_INDICATOR_OUT := TRUE;
		ELSE
			stateIdleCounter := stateIdleCounter + 1;
			IF(stateIdleCounter >= STATE_TIMEOUT) THEN
				stateIdleCounter := 0;
				state := SYSTEM_STATE.SYSTEM_READY;
			END_IF
		END_IF
		
END_CASE

END_PROGRAM

// ---- POUs/SYSTEM_RESET.TcPOU
PROGRAM SYSTEM_RESET
VAR CONSTANT
	TRANSITION_COUNT : INT := 10;
END_VAR

VAR
	cycleCounter : INT;
	state : RESET_STATE;
	
	ERROR_ACKNOWLEDGEMENT_BUTTON_OUT AT %Q* : BOOL;
	ESTOP_RESTART_BUTTON_OUT AT %Q* : BOOL;
END_VAR

IF GV_LIFT.SYSTEM_RESET_BUTTON_IN THEN
	cycleCounter := cycleCounter + 1;
	CASE state OF
		RESET_STATE.IDLE :
			IF(cycleCounter >= TRANSITION_COUNT) THEN
				state := RESET_STATE.ERRACK_ON;
				cycleCounter := 0;
			END_IF
		RESET_STATE.ERRACK_ON :
			ERROR_ACKNOWLEDGEMENT_BUTTON_OUT := TRUE;
			IF(cycleCounter >= TRANSITION_COUNT) THEN
				state := RESET_STATE.ERRACK_OFF;
				cycleCounter := 0;
			END_IF
		RESET_STATE.ERRACK_OFF :
			ERROR_ACKNOWLEDGEMENT_BUTTON_OUT := FALSE;
			IF(cycleCounter >= TRANSITION_COUNT) THEN
				state := RESET_STATE.IDLE2;
				cycleCounter := 0;
			END_IF
		RESET_STATE.IDLE2 :
			IF(cycleCounter >= TRANSITION_COUNT) THEN
				state := RESET_STATE.ESTOP_RESET_ON;
				cycleCounter := 0;
			END_IF
		RESET_STATE.ESTOP_RESET_ON :
			ESTOP_RESTART_BUTTON_OUT := TRUE;
			IF(cycleCounter >= TRANSITION_COUNT) THEN
				state := RESET_STATE.COMPLETE;
				cycleCounter := 0;
			END_IF
		RESET_STATE.COMPLETE :
			ESTOP_RESTART_BUTTON_OUT := FALSE;
	END_CASE
ELSE
	cycleCounter := 0;
	state := RESET_STATE.IDLE;
END_IF

END_PROGRAM

// ---- POUs/MOVE_TO_POSITION.TcPOU
PROGRAM MOVE_TO_POSITION
VAR CONSTANT
	UP_OFFSET : REAL :=-1.25;
	DOWN_OFFSET : REAL := 1.375;
	POSITION_SCALE : REAL := 12700;
	
END_VAR
VAR
	currentRawPosition AT %I* : UDINT;
	rStagePosition : REAL;
	rCurrentPosition : REAL;
	bRecalculatePosition : BOOL;
	WritePosCase : INT := 0;
END_VAR

rCurrentPosition := UDINT_TO_REAL(currentRawPosition);
CASE WritePosCase OF
0:	IF XML.LoadComplate THEN
		IF rStagePosition <> XML.savedvalues.rStagePosition THEN
			rStagePosition := XML.savedvalues.rStagePosition;
		END_IF
		WritePosCase := 1;
	ELSE rStagePosition := 2663040;
	END_IF
1:
	IF(bRecalculatePosition) THEN
		rStagePosition := rCurrentPosition - (POSITION_SCALE * GV_HMI.updatedPos);
			GV_LIFT.STAGE_POSITION := rStagePosition;
		bRecalculatePosition := FALSE;
	END_IF
	
	GV_LIFT.CURRENT_POSITION := (rCurrentPosition-rStagePosition)/ POSITION_SCALE;
	
	IF (GV_LIFT.RUN_BUTTON_OUT) AND GV_LIFT.MTS_ALLOWED	THEN
		IF(GV_LIFT.CURRENT_POSITION > (GV_LIFT.TARGET_POSITION + DOWN_OFFSET)) THEN
			GV_LIFT.DOWN_BUTTON_OUT := TRUE;
			GV_LIFT.JUST_RAN := TRUE;
		ELSIF(GV_LIFT.CURRENT_POSITION < (GV_LIFT.TARGET_POSITION + UP_OFFSET)) THEN
			GV_LIFT.UP_BUTTON_OUT := TRUE;
			GV_LIFT.JUST_RAN := TRUE;
		ELSE
			GV_LIFT.UP_BUTTON_OUT := FALSE;
			GV_LIFT.DOWN_BUTTON_OUT := FALSE;
			GV_LIFT.MTS_ALLOWED := FALSE;
			GV_LIFT.JUST_RAN:= FALSE;
		END_IF
	ELSIF GV_LIFT.JUST_RAN THEN
			GV_LIFT.MTS_ALLOWED := FALSE;
	END_IF

END_CASE

END_PROGRAM

// ---- POUs/Pendant Screen/SwitchScreens.TcPOU
PROGRAM SwitchScreens
VAR
	screenFound : BOOL := TRUE;
	screenSearchAttempts : INT := 0;
	screenRetryInerval: INT := 10;
	wasNoScreen : BOOL := FALSE;
	
	wasEstop : BOOL := FALSE;
	wasDoorFault : BOOL := FALSE;
	wasUpLimit : BOOL := FALSE;
	wasDwnLimit : BOOL := FALSE;
	wasJogging : BOOL := FALSE;
	wasRunningToTarget : BOOL := FALSE;
	doubleWrite : BOOL := FALSE;
	wasAcknowledge : BOOL := FALSE;
END_VAR

IF GV_MODBUS.screen.Error THEN
	screenFound := FALSE;
	wasNoScreen := TRUE;
	
	IF screenSearchAttempts > screenRetryInerval THEN
		screenFound := TRUE;
		GV_MODBUS.readExecute := TRUE;
	END_IF
	
	screenSearchAttempts := screenSearchAttempts + 1;
ELSE
	screenFound := TRUE;
		
	IF not GV_LIFT.ESTOP_INDICATOR_OUT THEN
		EStop();
		
		IF NOT wasEstop THEN
			Execute_Write_Screen();
		END_IF
		
		wasEstop := TRUE;
		GV_MODBUS.wasMTS := FALSE;
		wasDoorFault := FALSE;
		wasUpLimit := FALSE;
		wasDwnLimit := FALSE;
		wasJogging := FALSE;
		wasRunningToTarget := FALSE;
		wasAcknowledge := FALSE;
		
	ELSIF GV_LIFT.DOOR_1_INDICATOR_OUT OR GV_LIFT.DOOR_2_INDICATOR_OUT OR GV_LIFT.DOOR_3_INDICATOR_OUT OR GV_LIFT.DOOR_4_INDICATOR_OUT THEN	
		DoorFaults();	
	
		IF NOT wasDoorFault THEN
			Execute_Write_Screen();
		END_IF
		
		wasEstop := FALSE;
		GV_MODBUS.wasMTS := FALSE;
		wasDoorFault := TRUE;
		wasUpLimit := FALSE;
		wasDwnLimit := FALSE;
		wasJogging := FALSE;
		wasRunningToTarget := FALSE;
		wasAcknowledge := FALSE;
		
	ELSIF GV_LIFT.CRUSH_PROTECTION_INDICATOR_OUT THEN
		UpLimit();	
	
		IF NOT wasUpLimit THEN
			Execute_Write_Screen();
		END_IF
		
		wasEstop := FALSE;
		GV_MODBUS.wasMTS := FALSE;
		wasDoorFault := FALSE;
		wasUpLimit := TRUE;
		wasDwnLimit := FALSE;
		wasJogging := FALSE;
		wasRunningToTarget := FALSE;
		wasAcknowledge := FALSE;
		
	ELSIF (GV_LIFT.UP_LIMIT_INDICATOR_OUT OR GV_LIFT.CURRENT_POSITION > XML.savedvalues.UpSoftLim) AND NOT GV_MODBUS.limitAcknowledged THEN
		UpLimit();	
		
		IF NOT wasAcknowledge THEN
			Execute_Write_Screen();
		END_IF
		
		wasEstop := FALSE;
		GV_MODBUS.wasMTS := FALSE;
		wasDoorFault := FALSE;
		wasUpLimit := FALSE;
		wasDwnLimit := FALSE;
		wasJogging := FALSE;
		wasRunningToTarget := FALSE;
		wasAcknowledge := TRUE;
		
	ELSIF (GV_LIFT.ULTIMATE_LIMIT_INDICATOR_OUT OR GV_LIFT.DOWN_LIMIT_INDICATOR_OUT OR GV_LIFT.CURRENT_POSITION < XML.savedvalues.DownSoftLim) AND NOT GV_MODBUS.limitAcknowledged  THEN
		DownLimit();	
	
		IF NOT wasDwnLimit THEN
			Execute_Write_Screen();
		END_IF
		
		wasEstop := FALSE;
		GV_MODBUS.wasMTS := FALSE;
		wasDoorFault := FALSE;
		wasUpLimit := FALSE;
		wasDwnLimit := TRUE;
		wasJogging := FALSE;
		wasRunningToTarget := FALSE;
		wasAcknowledge := FALSE;
		
	ELSIF GV_LIFT.RUN_BUTTON_OUT AND GV_LIFT.MTS_ALLOWED THEN
		MoveToPosition();
		
		IF NOT wasRunningToTarget THEN
			Execute_Write_Screen();
		END_IF
		
		
		wasEstop := FALSE;
		GV_MODBUS.wasMTS := FALSE;
		wasDoorFault := FALSE;
		wasUpLimit := FALSE;
		wasDwnLimit := FALSE;
		wasJogging := FALSE;
		wasRunningToTarget := TRUE;
		wasAcknowledge := FALSE;
		
		GV_MODBUS.limitAcknowledged := FALSE;
	ELSIF GV_LIFT.UP_BUTTON_OUT OR GV_LIFT.DOWN_BUTTON_OUT THEN
		JogLift();
		
		IF NOT wasJogging THEN
			Execute_Write_Screen();	
		END_IF
		
		wasEstop := FALSE;
		GV_MODBUS.wasMTS := FALSE;
		wasDoorFault := FALSE;
		wasUpLimit := FALSE;
		wasDwnLimit := FALSE;
		wasJogging := TRUE;
		wasRunningToTarget := FALSE;
		wasAcknowledge := FALSE;
	
		GV_MODBUS.limitAcknowledged := FALSE;
	ELSE
		SelectSpike();
		
		IF NOT GV_MODBUS.wasMTS THEN
			Execute_Write_Screen();	
			doubleWrite := TRUE;		
		END_IF
		
		IF doubleWrite AND GV_MODBUS.doneWriting AND GV_MODBUS.wasMTS THEN
			Execute_Write_Screen();
			doubleWrite := FALSE;
		END_IF
		
		wasEstop := FALSE;
		GV_MODBUS.wasMTS := TRUE;
		wasDoorFault := FALSE;
		wasUpLimit := FALSE;
		wasDwnLimit := FALSE;
		wasJogging := FALSE;
		wasRunningToTarget := FALSE;
		wasAcknowledge := FALSE;
		
	END_IF
	
	IF wasNoScreen THEN
		wasNoScreen := FALSE;
		Execute_Write_Screen();
	END_IF
END_IF

IF screenFound THEN	
	ReadWriteScreen();
	screenSearchAttempts := 0;
END_IF

END_PROGRAM

// ---- POUs/Pendant Screen/EStop.TcPOU
PROGRAM EStop
VAR			
	estop_oneleft: ARRAY [1..5] OF WORD := [16#2A2A, 16#2A45, 16#4D45, 16#5247, 16#454E];
	estop_oneright: ARRAY [1..5] OF WORD := [16#4359, 16#2053, 16#544F, 16#502A, 16#2A2A];
	
	remote: ARRAY [1..5] OF WORD := [16#5265, 16#6D6F, 16#7465, 16#2020, 16#2020];
	pit: ARRAY [1..5] OF WORD := [16#5069, 16#7420, 16#2020, 16#2020, 16#2020];
	pump: ARRAY [1..5] OF WORD := [16#5075, 16#6D70, 16#2020, 16#2020, 16#2020];
	upstage: ARRAY [1..5] OF WORD := [16#5570, 16#7374, 16#6167, 16#6520, 16#2020];
	downstage: ARRAY [1..5] OF WORD := [16#446F, 16#776E, 16#7374, 16#6167, 16#6520];
	console: ARRAY [1..5] OF WORD := [16#436F, 16#6E73, 16#6F6C, 16#6520, 16#2020];
	
	pageNum: WORD := 0;	
END_VAR

IF GV_MODBUS.btnData = GV_MODBUS.btnUp THEN
	pageNum := 0;
	Execute_Write_Screen();
END_IF

IF GV_MODBUS.btnData = GV_MODBUS.btnDwn THEN
	pageNum := 1;
	Execute_Write_Screen();
END_IF

IF pageNum = 0 THEN
	GV_MODBUS.oneLeft:= estop_oneleft;
	GV_MODBUS.oneRight:= estop_oneright;   
                           
	GV_MODBUS.twoLeft:= remote;
	IF GV_LIFT.REMOTE_ESTOP_INDICATOR_OUT THEN
		GV_MODBUS.twoRight:= GV_MODBUS.engaged;
	ELSE
		GV_MODBUS.twoRight:= GV_MODBUS.ok;
	END_IF  
                            
	GV_MODBUS.threeLeft:= pit;
	IF GV_LIFT.PIT_ESTOP_INDICATOR_OUT THEN
		GV_MODBUS.threeRight:= GV_MODBUS.engaged;
	ELSE
		GV_MODBUS.threeRight:= GV_MODBUS.ok;
	END_IF	
                               
	GV_MODBUS.fourLeft:= pump; 
	IF GV_LIFT.PUMP_ESTOP_INDICATOR_OUT THEN
		GV_MODBUS.fourRight:= GV_MODBUS.engaged;
	ELSE
		GV_MODBUS.fourRight:= GV_MODBUS.ok;		
	END_IF
END_IF

IF pageNum = 1 THEN
	GV_MODBUS.oneLeft:= estop_oneleft;
	GV_MODBUS.oneRight:= estop_oneright;   
                           
	GV_MODBUS.twoLeft:= downstage;
	IF GV_LIFT.DOWNSTAGE_ESTOP_INDICATOR_OUT THEN
		GV_MODBUS.twoRight:= GV_MODBUS.engaged;
	ELSE
		GV_MODBUS.twoRight:= GV_MODBUS.ok;
	END_IF
                            
	GV_MODBUS.threeLeft:= upstage;
	IF GV_LIFT.UPSTAGE_ESTOP_INDICATOR_OUT THEN
		GV_MODBUS.threeRight:= GV_MODBUS.engaged;
	ELSE
		GV_MODBUS.threeRight:= GV_MODBUS.ok;
	END_IF
                               
	GV_MODBUS.fourLeft:= console; 
	IF GV_LIFT.CONSOLE_ESTOP_INDICATOR_OUT THEN
		GV_MODBUS.fourRight:= GV_MODBUS.engaged;
	ELSE
		GV_MODBUS.fourRight:= GV_MODBUS.ok;
	END_IF
END_IF

IF NOT GV_MODBUS.readExecute AND GV_MODBUS.addr = GV_MODBUS.oneLeftAddr THEN
	GV_MODBUS.data:= GV_MODBUS.oneLeft;
END_IF

END_PROGRAM

// ---- POUs/Pendant Screen/Functions/Execute_Write_Screen.TcPOU
FUNCTION Execute_Write_Screen : BOOL
VAR_INPUT
END_VAR
VAR
END_VAR

GV_MODBUS.addr := GV_MODBUS.oneLeftAddr;
GV_MODBUS.writeExecute := TRUE;
GV_MODBUS.readExecute := FALSE;
GV_MODBUS.doneWriting := FALSE;
GV_MODBUS.btnData := 0;

END_FUNCTION

// ---- POUs/Pendant Screen/DoorFaults.TcPOU
PROGRAM DoorFaults
VAR
	header_left : ARRAY [1..5] OF WORD := [16#2A2A, 16#2A2A, 16#2A44, 16#4F4F, 16#5220];
	header_right: ARRAY [1..5] OF WORD := [16#4641, 16#554C, 16#542A, 16#2A2A, 16#2A2A];
	
	usr_ok: ARRAY [1..5] OF WORD := [16#2055, 16#5352, 16#204F, 16#4B20, 16#2020];
	usr_fault: ARRAY [1..5] OF WORD := [16#2055, 16#5352, 16#2046, 16#4C54, 16#2020];
	                                   
	usl_ok: ARRAY [1..5] OF WORD := [16#2055, 16#534C, 16#204F, 16#4B20, 16#2020];
	usl_fault: ARRAY [1..5] OF WORD := [16#2055, 16#534C, 16#2046, 16#4C54, 16#2020];
	                                   
	dsr_ok: ARRAY [1..5] OF WORD := [16#2044, 16#5352, 16#204F, 16#4B20, 16#2020];
	dsr_fault: ARRAY [1..5] OF WORD := [16#2044, 16#5352, 16#2046, 16#4C54, 16#2020];
	                                   
	dsl_ok: ARRAY [1..5] OF WORD := [16#2044, 16#534C, 16#204F, 16#4B20, 16#2020];
	dsl_fault: ARRAY [1..5] OF WORD := [16#2044, 16#534C, 16#2046, 16#4C54, 16#2020];
	
	
	tick: INT := 0;
END_VAR

GV_MODBUS.oneLeft:= header_left;
GV_MODBUS.oneRight:= header_right;

GV_MODBUS.twoLeft:= GV_MODBUS.blank;
GV_MODBUS.twoRight:= GV_MODBUS.blank;

IF GV_LIFT.DOOR_1_INDICATOR_OUT THEN
	GV_MODBUS.threeLeft:= dsl_fault;
ELSE
	GV_MODBUS.threeLeft:= dsl_ok;
END_IF  

IF GV_LIFT.DOOR_2_INDICATOR_OUT THEN
	GV_MODBUS.threeRight:= dsr_fault;
ELSE
	GV_MODBUS.threeRight:= dsr_ok;
END_IF

IF GV_LIFT.DOOR_3_INDICATOR_OUT THEN
	GV_MODBUS.fourLeft:= usl_fault;
ELSE
	GV_MODBUS.fourLeft:= usl_ok;
END_IF

IF GV_LIFT.DOOR_4_INDICATOR_OUT THEN
	GV_MODBUS.fourRight:= usr_fault;
ELSE
	GV_MODBUS.fourRight:= usr_ok;
END_IF


IF tick >= GV_MODBUS.refreshInterval THEN
	Execute_Write_Screen();
	tick := 0;
END_IF

tick := tick + 1;

END_PROGRAM

// ---- POUs/Pendant Screen/UpLimit.TcPOU
PROGRAM UpLimit
VAR	
	crush_left : ARRAY [1..5] OF WORD := [16#2A2A, 16#2A2A, 16#2A43, 16#5255, 16#5348];
	crush_right : ARRAY [1..5] OF WORD := [16#2046, 16#4155, 16#4C54, 16#2A2A, 16#2A2A];
	
	hard_left : ARRAY [1..5] OF WORD := [16#2A2A, 16#2A2A, 16#5550, 16#2048, 16#4152];
	hard_right : ARRAY [1..5] OF WORD := [16#4420, 16#4C49, 16#4D49, 16#542A, 16#2A2A];
	
	soft_left : ARRAY [1..5] OF WORD := [16#2A2A, 16#2A2A, 16#5550, 16#2053, 16#4F46];
	soft_right : ARRAY [1..5] OF WORD := [16#5420, 16#4C49, 16#4D49, 16#542A, 16#2A2A];	
	
	crush_message_left : ARRAY [1..5] OF WORD := [16#2020, 16#504C, 16#4541, 16#5345, 16#204A];
	crush_message_right : ARRAY [1..5] OF WORD := [16#4F47, 16#2044, 16#4F57, 16#4E20, 16#2020];
	
	message_left : ARRAY [1..5] OF WORD := [16#2050, 16#5245, 16#5353, 16#2053, 16#454C];
	message_right : ARRAY [1..5] OF WORD := [16#4543, 16#5420, 16#2F20, 16#4A4F, 16#4720];
	
	current : ARRAY [1..5] OF WORD := [16#4375, 16#7272, 16#656E, 16#7420, 16#506F];
	pos : ARRAY [1..5] OF WORD := [16#7320, 16#2020, 16#2020, 16#2020, 16#2020];
	tick: INT := 0;
END_VAR

IF GV_MODBUS.btnData = GV_MODBUS.btnEnter THEN
	GV_MODBUS.limitAcknowledged := TRUE;
END_IF

GV_MODBUS.twoLeft:= message_left;
GV_MODBUS.twoRight:= message_right;

IF GV_LIFT.CRUSH_PROTECTION_INDICATOR_OUT THEN
	GV_MODBUS.oneLeft := crush_left;
	GV_MODBUS.oneRight := crush_right;
	
	GV_MODBUS.twoLeft:= crush_message_left;
	GV_MODBUS.twoRight:= crush_message_right;
ELSIF GV_LIFT.UP_LIMIT_INDICATOR_OUT THEN
	GV_MODBUS.oneLeft := hard_left;
	GV_MODBUS.oneRight := hard_right;
ELSIF GV_LIFT.CURRENT_POSITION > XML.savedvalues.UpSoftLim THEN
	GV_MODBUS.oneLeft := soft_left;
	GV_MODBUS.oneRight := soft_right;
END_IF

GV_MODBUS.threeLeft := GV_MODBUS.blank;
GV_MODBUS.threeRight := GV_MODBUS.blank;

GV_MODBUS.fourLeft:= current;
GV_MODBUS.fourRight:= GV_MODBUS.blank;	

GV_MODBUS.fourRight:= Position_To_Row_Array(pos, GV_LIFT.CURRENT_POSITION);     


IF tick >= (GV_MODBUS.refreshInterval*2) THEN
	Execute_Write_Screen();
	tick := 0;
END_IF

tick := tick + 1;

END_PROGRAM

// ---- POUs/Pendant Screen/Functions/Position_To_Row_Array.TcPOU
FUNCTION Position_To_Row_Array : ARRAY[1..5] OF WORD
VAR_INPUT
	row: ARRAY[1..5] OF WORD;
	position: REAL;
END_VAR
VAR
	posLen: INT;
	posString: STRING;
	n:BYTE:=8;
END_VAR

posString := LREAL_TO_FMTSTR(position, 1, TRUE);
posLen := LEN(posString);
	
IF posLen = 3 THEN
	row[3] := row[3] AND 16#FF00;
	row[3] :=  row[3] OR GV_MODBUS.space;
	
	row[4] := posString[0];
	row[4] := SHL(row[4], n);
	row[4] := row[4] OR posString[1];
	
	row[5] := posString[2];
	row[5] := SHL(row[5], n);
	row[5] := row[5] OR GV_MODBUS.inch;
END_IF

IF posLen = 4 THEN
	
	row[3] := GV_MODBUS.space;
	row[3] := SHL(row[3], n);
	row[3] := row[3] OR posString[0];
	
	row[4] := posString[1];
	row[4] := SHL(row[4], n);
	row[4] := row[4] OR posString[2];
	
	row[5] := posString[3];
	row[5] := SHL(row[5], n);
	row[5] := row[5] OR GV_MODBUS.inch;
END_IF

IF posLen = 5 THEN
	
	row[2] := row[2] AND 16#FF00;	
	row[2] := row[2] OR GV_MODBUS.space;
	
	row[3] := posString[0];
	row[3] := SHL(row[3], n);
	row[3] := row[3] OR posString[1];
		
	row[4] := posString[2];
	row[4] := SHL(row[4], n);
	row[4] := row[4] OR posString[3];
		
	row[5] := posString[4];
	row[5] := SHL(row[5], n);
	row[5] := row[5] OR GV_MODBUS.inch;
	
END_IF

IF posLen = 6 THEN
	row[2] := GV_MODBUS.space;	
	row[2] := SHL(row[2], n);
	row[2] := row[2] OR posString[0];
	 
	row[3] := posString[1];
	row[3] := SHL(row[3], n);
	row[3] := row[3] OR posString[2];
	 
	row[4] := posString[3];
	row[4] := SHL(row[4], n);
	row[4] := row[4] OR posString[4];
	 
	row[5] := posString[5];
	row[5] := SHL(row[5], n);
	row[5] := row[5] OR GV_MODBUS.inch;
	
END_IF

Position_To_Row_Array := row;

END_FUNCTION

// ---- POUs/Pendant Screen/DownLimit.TcPOU
PROGRAM DownLimit
VAR	
	ult_left : ARRAY [1..5] OF WORD := [16#2A2A, 16#2A44, 16#4F57, 16#4E20, 16#554C];
	ult_right : ARRAY [1..5] OF WORD := [16#5420, 16#4C49, 16#4D49, 16#542A, 16#2A2A];

	hard_left : ARRAY [1..5] OF WORD := [16#2A2A, 16#2A44, 16#4F57, 16#4E20, 16#4841];
	hard_right : ARRAY [1..5] OF WORD := [16#5244, 16#204C, 16#494D, 16#4954, 16#2A2A];

	soft_left : ARRAY [1..5] OF WORD := [16#2A2A, 16#2A44, 16#4F57, 16#4E20, 16#534F];
	soft_right : ARRAY [1..5] OF WORD := [16#4654, 16#204C, 16#494D, 16#4954, 16#2A2A];
		

	//message_left : ARRAY [1..5] OF WORD := [16#2020, 16#2050, 16#4C45, 16#4153, 16#4520];
	//message_right : ARRAY [1..5] OF WORD := [16#4A4F, 16#4720, 16#5550, 16#2020, 16#2020];	
	message_left : ARRAY [1..5] OF WORD := [16#2050, 16#5245, 16#5353, 16#2053, 16#454C];
	message_right : ARRAY [1..5] OF WORD := [16#4543, 16#5420, 16#2F20, 16#4A4F, 16#4720];
	
	current : ARRAY [1..5] OF WORD := [16#4375, 16#7272, 16#656E, 16#7420, 16#506F];
	pos : ARRAY [1..5] OF WORD := [16#7320, 16#2020, 16#2020, 16#2020, 16#2020];
	
	tick: INT := 0;
END_VAR

IF GV_MODBUS.btnData = GV_MODBUS.btnEnter THEN
	GV_MODBUS.limitAcknowledged := TRUE;
END_IF

GV_MODBUS.twoLeft:= message_left;
GV_MODBUS.twoRight:= message_right;

IF GV_LIFT.ULTIMATE_LIMIT_INDICATOR_OUT THEN
	GV_MODBUS.oneLeft := ult_left;
	GV_MODBUS.oneRight := ult_right;
ELSIF GV_LIFT.DOWN_LIMIT_INDICATOR_OUT THEN
	GV_MODBUS.oneLeft := hard_left;
	GV_MODBUS.oneRight := hard_right;
ELSIF GV_LIFT.CURRENT_POSITION < XML.savedvalues.DownSoftLim THEN
	GV_MODBUS.oneLeft := soft_left;
	GV_MODBUS.oneRight := soft_right;
END_IF

GV_MODBUS.threeLeft := GV_MODBUS.blank;
GV_MODBUS.threeRight := GV_MODBUS.blank;

GV_MODBUS.fourLeft:= current;
GV_MODBUS.fourRight:= GV_MODBUS.blank;	

GV_MODBUS.fourRight:= Position_To_Row_Array(pos, GV_LIFT.CURRENT_POSITION);     


IF tick >= (GV_MODBUS.refreshInterval*2) THEN
	Execute_Write_Screen();
	tick := 0;
END_IF

tick := tick + 1;

END_PROGRAM

// ---- POUs/Pendant Screen/MoveToPosition.TcPOU
PROGRAM MoveToPosition
VAR
	mtpOneLeft : ARRAY[1..5] OF WORD := [16#2A2A, 16#4D4F, 16#5645, 16#2054, 16#4F20];
	mtpOneRight : ARRAY[1..5] OF WORD := [16#504F, 16#5349, 16#5449, 16#4F4E, 16#2A2A];
	
	current : ARRAY[1..5] OF WORD := [16#4375, 16#7272, 16#656E, 16#7420, 16#506F];
	target : ARRAY[1..5] OF WORD := [16#5461, 16#7267, 16#6574, 16#2020, 16#506F];
	pos : ARRAY[1..5] OF WORD := [16#7320, 16#2020, 16#2020, 16#2020, 16#2020];
	
	tick : INT := 0;
END_VAR

GV_MODBUS.oneLeft:= mtpOneLeft;         
GV_MODBUS.oneRight:= mtpOneRight;

GV_MODBUS.twoLeft:= GV_MODBUS.blank; 
GV_MODBUS.twoRight:= GV_MODBUS.blank;


GV_MODBUS.threeLeft:= current;
GV_MODBUS.threeRight:= GV_MODBUS.blank;
GV_MODBUS.threeRight:= Position_To_Row_Array(pos, GV_LIFT.CURRENT_POSITION);     

GV_MODBUS.fourLeft:= target;
GV_MODBUS.fourRight:= GV_MODBUS.blank;	
GV_MODBUS.fourRight:= Position_To_Row_Array(pos, GV_LIFT.TARGET_POSITION);

IF tick >= GV_MODBUS.refreshInterval THEN
	Execute_Write_Screen();
	tick := 0;
END_IF

tick := tick + 1;

END_PROGRAM

// ---- POUs/Pendant Screen/JogLift.TcPOU
PROGRAM JogLift
VAR
	jogOneLeft : ARRAY [1..5] OF WORD := [16#2A2A, 16#2A2A, 16#2A2A, 16#4A4F, 16#4720];
	jogOneRight : ARRAY [1..5] OF WORD := [16#4C49, 16#4654, 16#2A2A, 16#2A2A, 16#2A2A];
	current : ARRAY [1..5] OF WORD := [16#4375, 16#7272, 16#656E, 16#7420, 16#506F];
	pos : ARRAY [1..5] OF WORD := [16#7320, 16#2020, 16#2020, 16#2020, 16#2020];
	moving : ARRAY [1..5] OF WORD := [16#4D6F, 16#7669, 16#6E67, 16#2020, 16#2020];
	up : ARRAY [1..5] OF WORD := [16#2020, 16#2020, 16#2020, 16#2020, 16#5570];
	down : ARRAY [1..5] OF WORD := [16#2020, 16#2020, 16#2020, 16#446F, 16#776E];
	
	movingUpLeft : ARRAY [1..5] OF WORD := [16#2A2A, 16#2A4A, 16#4F47, 16#204C, 16#4946];
	movingUpRight : ARRAY [1..5] OF WORD := [16#5420, 16#2D20, 16#5550, 16#2A2A, 16#2A2A];
	movingDownLeft : ARRAY [1..5] OF WORD := [16#2A2A, 16#2A4A, 16#4F47, 16#204C, 16#4946];
	movingDownRight : ARRAY [1..5] OF WORD := [16#5420, 16#2D20, 16#444E, 16#2A2A, 16#2A2A];
	
	allowedToMove : BOOL := FALSE;
	tick : INT := 0;
END_VAR

GV_MODBUS.oneLeft:= GV_MODBUS.blank;         
GV_MODBUS.oneRight:= GV_MODBUS.blank;

GV_MODBUS.twoLeft:= GV_MODBUS.blank;
GV_MODBUS.twoRight:= GV_MODBUS.blank;

GV_MODBUS.threeLeft:= current;
GV_MODBUS.threeRight:= GV_MODBUS.blank;	

GV_MODBUS.fourLeft:= GV_MODBUS.blank; 
GV_MODBUS.fourRight:= GV_MODBUS.blank;

GV_MODBUS.threeRight:= Position_To_Row_Array(pos, GV_LIFT.CURRENT_POSITION);     

IF GV_LIFT.DOWN_BUTTON_OUT THEN
	GV_MODBUS.oneLeft:= movingDownLeft;
	GV_MODBUS.oneRight := movingDownRight;
ELSE
	GV_MODBUS.oneLeft:= movingUpLeft;
	GV_MODBUS.oneRight := movingUpRight;
END_IF

IF tick >= GV_MODBUS.refreshInterval THEN
	Execute_Write_Screen();
	tick := 0;
END_IF

tick := tick + 1;

END_PROGRAM

// ---- POUs/Pendant Screen/SelectSpike.TcPOU
PROGRAM SelectSpike
VAR
	current_pos: ARRAY [1..5] OF WORD :=[16#4355, 16#5252, 16#454E, 16#5420, 16#504F];
	pos: ARRAY [1..5] OF WORD := [16#5320, 16#2020, 16#2020, 16#2020, 16#2020];

	row: ARRAY [1..10] OF WORD;
	indexs: ARRAY [1..GV_HMI.iMaxTargets] OF INT;
	found: BOOL := FALSE;
	
	indexesIndex: INT := 1;
	firstSpikeIndex: INT := 0;
	secondSpikeIndex: INT := 0;
	thirdSpikeIndex: INT := 0;	
	
	selectedCursorIndex: INT := 0;	
	cursorIndex: INT := 1;
	lastPos : REAL := GV_LIFT.TARGET_POSITION;
	noneSelectedTargetPosValue : REAL := 0;
	tempTarget : REAL := 0;
	
	maxCursorIndex : INT := 0;
END_VAR

indexs := Get_Valid_Indexs();

IF GV_MODBUS.btnData = GV_MODBUS.btnUp THEN
	cursorIndex:= cursorIndex - 1;
	selectedCursorIndex := 0;
	GV_LIFT.MTS_ALLOWED := FALSE;
	GV_LIFT.JUST_RAN := FALSE;
	Execute_Write_Screen();
END_IF

IF GV_MODBUS.btnData = GV_MODBUS.btnDwn THEN
	cursorIndex:= cursorIndex + 1;	
	selectedCursorIndex := 0;
	GV_LIFT.MTS_ALLOWED := FALSE;
	GV_LIFT.JUST_RAN := FALSE;
	Execute_Write_Screen();	
END_IF

IF NOT GV_MODBUS.wasMTS THEN
	selectedCursorIndex := 0;
	//GV_LIFT.TARGET_POSITION := noneSelectedTargetPosValue;
END_IF

IF (indexs[3] > 0) THEN
	maxCursorIndex := 3;
ELSIF(indexs[2] > 0) THEN 
	maxCursorIndex := 2;
ELSIF(indexs[1] > 0) THEN
	maxCursorIndex := 1;
ELSE
	maxCursorIndex := 0;
END_IF


IF GV_MODBUS.btnData = GV_MODBUS.btnEnter THEN
	selectedCursorIndex := cursorIndex;
	
	IF cursorIndex = 1 THEN
		tempTarget := XML.savedvalues.savedpos[firstSpikeIndex].target;
	ELSIF cursorIndex = 2 THEN
		tempTarget := XML.savedvalues.savedpos[secondSpikeIndex].target;
	ELSIF cursorIndex = 3 THEN
		tempTarget := XML.savedvalues.savedpos[thirdSpikeIndex].target;
	END_IF
	
	IF tempTarget >=  XML.savedvalues.DownSoftLim AND tempTarget <=  XML.savedvalues.UpSoftLim THEN
		GV_LIFT.MTS_ALLOWED := TRUE;
		GV_LIFT.JUST_RAN := FALSE;
		GV_LIFT.TARGET_POSITION := tempTarget;
	END_IF	
	
	Execute_Write_Screen();
END_IF

IF firstSpikeIndex = 0 THEN
	firstSpikeIndex := indexs[1];
	secondSpikeIndex := indexs[2];
	thirdSpikeIndex := indexs[3];
END_IF

IF cursorIndex < 1 THEN
	indexesIndex := indexesIndex - 1;
	
	IF indexesIndex < 1 THEN
		indexesIndex := 1;
	END_IF
	
	firstSpikeIndex := indexs[indexesIndex];
	secondSpikeIndex := indexs[indexesIndex + 1];
	thirdSpikeIndex := indexs[indexesIndex + 2];
	
	cursorIndex := 1;
END_IF

IF cursorIndex > maxCursorIndex THEN	
	indexesIndex := indexesIndex + 1;
	
	IF indexesIndex > (GV_HMI.iMaxTargets - 2) THEN
		indexesIndex := GV_HMI.iMaxTargets - 2;
	END_IF
	
	IF indexs[indexesIndex + 2] = 0 THEN
		indexesIndex := indexesIndex - 1;
	END_IF
	
	IF indexesIndex < 1 THEN
		indexesIndex := 1;
	END_IF
		
	firstSpikeIndex := indexs[indexesIndex];
	secondSpikeIndex := indexs[indexesIndex + 1];
	thirdSpikeIndex := indexs[indexesIndex + 2];
	
	cursorIndex := maxCursorIndex;
END_IF

GV_MODBUS.oneLeft:= current_pos;         
GV_MODBUS.oneRight:= GV_MODBUS.blank;
GV_MODBUS.twoLeft:= GV_MODBUS.blank;
GV_MODBUS.twoRight:= GV_MODBUS.blank;
GV_MODBUS.threeLeft:= GV_MODBUS.blank;
GV_MODBUS.threeRight:= GV_MODBUS.blank;	
GV_MODBUS.fourLeft:= GV_MODBUS.blank; 
GV_MODBUS.fourRight:= GV_MODBUS.blank;

GV_MODBUS.oneRight:= Position_To_Row_Array(pos, GV_LIFT.CURRENT_POSITION);     
	
IF firstSpikeIndex > 0 THEN		
	IF XML.savedvalues.savedpos[firstSpikeIndex].target < GV_MODBUS.filterTarget THEN
		
		
		IF cursorIndex = 1 AND NOT (selectedCursorIndex = 1) THEN
			row := Spike_To_Row_Array(GV_MODBUS.selectedASCII, XML.savedvalues.savedpos[firstSpikeIndex]);
		ELSIF selectedCursorIndex = 1 AND GV_LIFT.MTS_ALLOWED THEN
			row := Spike_To_Row_Array(GV_MODBUS.loadedASCII, XML.savedvalues.savedpos[firstSpikeIndex]);
		ELSIF selectedCursorIndex = 1 AND NOT GV_LIFT.MTS_ALLOWED THEN			
			row := Spike_To_Row_Array(GV_MODBUS.outOfBoundsASCII, XML.savedvalues.savedpos[firstSpikeIndex]);
		ELSE
			row := Spike_To_Row_Array(GV_MODBUS.spaceASCII, XML.savedvalues.savedpos[firstSpikeIndex]);
		END_IF
		
		Fill_Row_Two(row);
	END_IF
END_IF
	
IF secondSpikeIndex > 0 THEN					   
	IF XML.savedvalues.savedpos[secondSpikeIndex].target < GV_MODBUS.filterTarget THEN
		
		
		IF cursorIndex = 2 AND NOT (selectedCursorIndex = 2) THEN
			row := Spike_To_Row_Array(GV_MODBUS.selectedASCII, XML.savedvalues.savedpos[secondSpikeIndex]);		
		ELSIF selectedCursorIndex = 2  AND GV_LIFT.MTS_ALLOWED THEN
			row := Spike_To_Row_Array(GV_MODBUS.loadedASCII, XML.savedvalues.savedpos[secondSpikeIndex]);	
		ELSIF selectedCursorIndex = 2 AND NOT GV_LIFT.MTS_ALLOWED THEN
			row := Spike_To_Row_Array(GV_MODBUS.outOfBoundsASCII, XML.savedvalues.savedpos[secondSpikeIndex]);				
		ELSE
			row := Spike_To_Row_Array(GV_MODBUS.spaceASCII, XML.savedvalues.savedpos[secondSpikeIndex]);
		END_IF
		 
		Fill_Row_Three(row);
	END_IF	
END_IF

IF thirdSpikeIndex > 0 THEN
	IF XML.savedvalues.savedpos[thirdSpikeIndex].target < GV_MODBUS.filterTarget THEN
		IF cursorIndex = 3 AND NOT (selectedCursorIndex = 3) THEN
			row := Spike_To_Row_Array(GV_MODBUS.selectedASCII, XML.savedvalues.savedpos[thirdSpikeIndex]); 				
		ELSIF selectedCursorIndex = 3 AND GV_LIFT.MTS_ALLOWED THEN
			row := Spike_To_Row_Array(GV_MODBUS.loadedASCII, XML.savedvalues.savedpos[thirdSpikeIndex]);
		ELSIF selectedCursorIndex = 3 AND NOT GV_LIFT.MTS_ALLOWED THEN
			row := Spike_To_Row_Array(GV_MODBUS.outOfBoundsASCII, XML.savedvalues.savedpos[thirdSpikeIndex]);			
		ELSE
			row := Spike_To_Row_Array(GV_MODBUS.spaceASCII, XML.savedvalues.savedpos[thirdSpikeIndex]); 
		END_IF
		
		Fill_Row_Four(row);				
	END_IF
END_IF

IF NOT GV_MODBUS.readExecute AND GV_MODBUS.addr = GV_MODBUS.oneLeftAddr THEN
	GV_MODBUS.data:= GV_MODBUS.oneLeft;
END_IF

END_PROGRAM

// ---- POUs/Pendant Screen/Functions/Get_Valid_Indexs.TcPOU
FUNCTION Get_Valid_Indexs : ARRAY [1..GV_HMI.iMaxTargets] OF INT
VAR_INPUT
END_VAR
VAR
	indexes: ARRAY [1..GV_HMI.iMaxTargets] OF INT;
	i: INT;
	j: INT;
END_VAR

j := 1;
FOR i:=1 TO GV_HMI.iMaxTargets BY 1 DO 
   IF XML.savedvalues.savedpos[i].targetclear THEN
	   indexes[j] := i;
	   j := j + 1;
   END_IF
END_FOR;

Get_Valid_Indexs := indexes;

END_FUNCTION

// ---- POUs/Pendant Screen/Functions/Spike_To_Row_Array.TcPOU
FUNCTION Spike_To_Row_Array : ARRAY [1..10] OF WORD
VAR_INPUT
	firstChar: STRING;
	spike: ST_SavedPositions;
END_VAR
VAR	
	left: ARRAY [1..5] OF WORD;
	right: ARRAY[1..5] OF WORD;
	rightPosition: ARRAY[1..5] OF WORD;
	
	spikeName: STRING;
	
END_VAR

spikeName := CONCAT(firstChar, spike.description);

left:= Spike_To_Half_Row_Array(MID(spikeName, 10, 1));
right:= Spike_To_Half_Row_Array(MID(spikeName, 10, 11));

rightPosition:= Position_To_Row_Array(right, spike.target);

Spike_To_Row_Array[1] := left[1];
Spike_To_Row_Array[2] := left[2];
Spike_To_Row_Array[3] := left[3];
Spike_To_Row_Array[4] := left[4];
Spike_To_Row_Array[5] := left[5];
Spike_To_Row_Array[6] := rightPosition[1];
Spike_To_Row_Array[7] := rightPosition[2];
Spike_To_Row_Array[8] := rightPosition[3];
Spike_To_Row_Array[9] := rightPosition[4];
Spike_To_Row_Array[10] := rightPosition[5];

END_FUNCTION

// ---- POUs/Pendant Screen/Functions/Spike_To_Half_Row_Array.TcPOU
FUNCTION Spike_To_Half_Row_Array : ARRAY[1..5] OF WORD
VAR_INPUT
	spikeName: String;	
END_VAR
VAR
	row: ARRAY[1..5] OF WORD;
	n:BYTE:=8;
	spikeNameLen: INT := 0;
	
	spikeIndex: INT := 0;
	rowIndex: INT := 1;
END_VAR

spikeIndex := 0;
rowIndex := 1;
spikeNameLen := LEN(spikeName);
row:= GV_MODBUS.blank;

WHILE rowIndex < 6 DO	
	IF spikeIndex < spikeNameLen  THEN
		row[rowIndex] := spikeName[spikeIndex];
	ELSE
		row[rowIndex] := GV_MODBUS.space;
	END_IF	
	row[rowIndex] := SHL(row[rowIndex], n);		
	spikeIndex := spikeIndex + 1;
	
	IF spikeIndex < spikeNameLen THEN
		row[rowIndex] := row[rowIndex] OR spikeName[spikeIndex];
	ELSE
		row[rowIndex] := row[rowIndex] OR GV_MODBUS.space;		
	END_IF
	spikeIndex := spikeIndex + 1;
	
	rowIndex := rowIndex + 1;	
END_WHILE

Spike_To_Half_Row_Array := row;

END_FUNCTION

// ---- POUs/Pendant Screen/Functions/Fill_Row_Two.TcPOU
FUNCTION Fill_Row_Two : BOOL
VAR_INPUT
	row: ARRAY [1..10] OF WORD;
END_VAR
VAR
END_VAR

GV_MODBUS.twoLeft[1]:= row[1];
GV_MODBUS.twoLeft[2]:= row[2];
GV_MODBUS.twoLeft[3]:= row[3];
GV_MODBUS.twoLeft[4]:= row[4];
GV_MODBUS.twoLeft[5]:= row[5];
GV_MODBUS.twoRight[1]:= row[6];
GV_MODBUS.twoRight[2]:= row[7];
GV_MODBUS.twoRight[3]:= row[8];
GV_MODBUS.twoRight[4]:= row[9];
GV_MODBUS.twoRight[5]:= row[10];

Fill_Row_Two := TRUE;

END_FUNCTION

// ---- POUs/Pendant Screen/Functions/Fill_Row_Three.TcPOU
FUNCTION Fill_Row_Three : BOOL
VAR_INPUT
	row: ARRAY[1..10] OF WORD;
END_VAR
VAR
END_VAR

GV_MODBUS.threeLeft[1]:= row[1];
GV_MODBUS.threeLeft[2]:= row[2];
GV_MODBUS.threeLeft[3]:= row[3];
GV_MODBUS.threeLeft[4]:= row[4];
GV_MODBUS.threeLeft[5]:= row[5];
GV_MODBUS.threeRight[1]:= row[6];
GV_MODBUS.threeRight[2]:= row[7];
GV_MODBUS.threeRight[3]:= row[8];
GV_MODBUS.threeRight[4]:= row[9];
GV_MODBUS.threeRight[5]:= row[10];

END_FUNCTION

// ---- POUs/Pendant Screen/Functions/Fill_Row_Four.TcPOU
FUNCTION Fill_Row_Four : BOOL
VAR_INPUT
	row: ARRAY[1..10] OF WORD;
END_VAR
VAR
END_VAR

GV_MODBUS.fourLeft[1]:= row[1];
GV_MODBUS.fourLeft[2]:= row[2];
GV_MODBUS.fourLeft[3]:= row[3];
GV_MODBUS.fourLeft[4]:= row[4];
GV_MODBUS.fourLeft[5]:= row[5];
GV_MODBUS.fourRight[1]:= row[6];
GV_MODBUS.fourRight[2]:= row[7];
GV_MODBUS.fourRight[3]:= row[8];
GV_MODBUS.fourRight[4]:= row[9];
GV_MODBUS.fourRight[5]:= row[10];

END_FUNCTION

// ---- POUs/Pendant Screen/ReadWriteScreen.TcPOU
PROGRAM ReadWriteScreen
VAR
	writeBusy: BOOL;
	writeError: BOOL;
	writeErrorId: MODBUS_ERRORS;
	readBusy: BOOL;
	readError: BOOL;
	readErrorId: MODBUS_ERRORS;	
END_VAR

GV_MODBUS.screen.WriteRegs(
	UnitID:= GV_MODBUS.UnitID, 
	Timeout:= GV_MODBUS.timeout,
	Quantity:= GV_MODBUS.quantity,
	cbLength:= GV_MODBUS.quantity * 2,
	Execute:= GV_MODBUS.writeExecute,
	MBAddr := GV_MODBUS.addr,
	pMemoryAddr:= ADR(GV_MODBUS.data),
	Busy=> writeBusy,
	Error=> writeError,
	ErrorId=> writeErrorId
);	

GV_MODBUS.writeExecute := FALSE;

GV_MODBUS.screen.ReadRegs(
	UnitID:= GV_MODBUS.UnitID, 
	Timeout:= GV_MODBUS.timeout,
	Quantity:= 1,
	cbLength:= 2,
	Execute:= GV_MODBUS.readExecute,
	MBAddr := 16#3A,
	pMemoryAddr:= ADR(GV_MODBUS.btnData),
	Busy=> readBusy,
	Error=> readError,
	ErrorId=> readErrorId
);	

IF NOT GV_MODBUS.screen.Busy THEN 
	IF GV_MODBUS.screen.Error THEN 
		GV_MODBUS.addr:= 99;
	ELSE 
		IF GV_MODBUS.doneWriting THEN
			GV_MODBUS.addr := GV_MODBUS.oneLeftAddr;
			GV_MODBUS.data:= GV_MODBUS.oneLeft;
			GV_MODBUS.readExecute := TRUE;	
		ELSIF GV_MODBUS.addr = GV_MODBUS.oneLeftAddr THEN
			GV_MODBUS.addr := GV_MODBUS.oneRightAddr;
			GV_MODBUS.data:= GV_MODBUS.oneRight;
			GV_MODBUS.writeExecute := TRUE;
		ELSIF GV_MODBUS.addr = GV_MODBUS.oneRightAddr THEN
			GV_MODBUS.addr := GV_MODBUS.twoLeftAddr;
			GV_MODBUS.data:= GV_MODBUS.twoLeft;
			GV_MODBUS.writeExecute := TRUE;
		ELSIF GV_MODBUS.addr = GV_MODBUS.twoLeftAddr THEN
			GV_MODBUS.addr := GV_MODBUS.twoRightAddr;
			GV_MODBUS.data:= GV_MODBUS.twoRight;
			GV_MODBUS.writeExecute := TRUE;
		ELSIF GV_MODBUS.addr = GV_MODBUS.twoRightAddr THEN
			GV_MODBUS.addr := GV_MODBUS.threeLeftAddr;
			GV_MODBUS.data:= GV_MODBUS.threeLeft;
			GV_MODBUS.writeExecute := TRUE;
		ELSIF GV_MODBUS.addr = GV_MODBUS.threeLeftAddr THEN
			GV_MODBUS.addr := GV_MODBUS.threeRightAddr;
			GV_MODBUS.data:= GV_MODBUS.threeRight;
			GV_MODBUS.writeExecute := TRUE;
		ELSIF GV_MODBUS.addr = GV_MODBUS.threeRightAddr THEN
			GV_MODBUS.addr := GV_MODBUS.fourLeftAddr;
			GV_MODBUS.data:= GV_MODBUS.fourLeft;
			GV_MODBUS.writeExecute := TRUE;
		ELSIF GV_MODBUS.addr = GV_MODBUS.fourLeftAddr THEN
			GV_MODBUS.addr := GV_MODBUS.fourRightAddr;
			GV_MODBUS.data:= GV_MODBUS.fourRight;
			GV_MODBUS.writeExecute := TRUE;
		ELSIF GV_MODBUS.addr = GV_MODBUS.fourRightAddr THEN
			GV_MODBUS.addr := GV_MODBUS.oneLeftAddr;
			GV_MODBUS.data:= GV_MODBUS.oneLeft;
			GV_MODBUS.writeExecute := TRUE;
			GV_MODBUS.doneWriting := TRUE;
		END_IF		
	END_IF
END_IF

END_PROGRAM

// ---- GlobalTextList.TcGTLO
TEXTLIST GlobalTextList
  866 = '%.2f'
  166 = '%.2f"'
  559 = '%.3f"'
  982 = '%f"'
  24 = '%s'
  742 = '%s"'
  747 = 'Clear Target'
  136 = 'Console E-Stop'
  142 = 'Crush Detected'
  143 = 'Crush Protection'
  741 = 'current position:'
  537 = 'DELETE TARGET'
  75 = 'Delete Target'
  423 = 'Desciption'
  516 = 'Description'
  300 = 'Door 1 - DSL'
  132 = 'Door 2 - DSR'
  133 = 'Door 3 - USL'
  134 = 'Door 4 - USR'
  439 = 'Door Interlock'
  135 = 'Door Interlocks'
  298 = 'DOWN EOT Limit'
  532 = 'DOWN Hard Limit'
  297 = 'DOWN Soft Limit'
  990 = 'DOWN Soft Limit: %.2f"'
  944 = 'DOWN ULT Limit'
  255 = 'DOWN ultimate Limit'
  725 = 'DOWN Ultimate Limit'
  141 = 'DS Door E-Stop'
  436 = 'E-STOP'
  307 = 'EDIT'
  599 = 'Edit Description'
  748 = 'EDIT MODE:'
  598 = 'Edit Target Position'
  641 = 'EDIT TARGETS'
  140 = 'Emergency Stop'
  437 = 'EOT Limit'
  79 = 'Hard Limit'
  299 = 'Limit Status'
  744 = 'Load Target'
  572 = 'Pendant E-Stop'
  138 = 'Pickle E-Stop'
  137 = 'Pit E-Stop'
  736 = 'Properties'
  839 = 'Pump Room E-Stop'
  376 = 'RUN'
  746 = 'Safety Status Panel'
  144 = 'Set Current Position'
  146 = 'Set DOWN Soft Limit'
  145 = 'Set UP Soft Limit'
  438 = 'Soft Limit'
  435 = 'SYSTEM'
  440 = 'System Fault'
  638 = 'Target'
  571 = 'Target Position'
  743 = 'target position:'
  745 = 'Target Positions'
  162 = 'Unload Target'
  483 = 'UP End Of Travel Limit'
  295 = 'UP EOT Limit'
  446 = 'UP Hard Limit'
  296 = 'UP Soft Limit'
  453 = 'UP Soft Limit %.2f"'
  139 = 'US Door E-Stop'
  103 = 'Write XML'
END_TEXTLIST

// ---- VISUs/MAIN_DASHBOARD.TcVIS
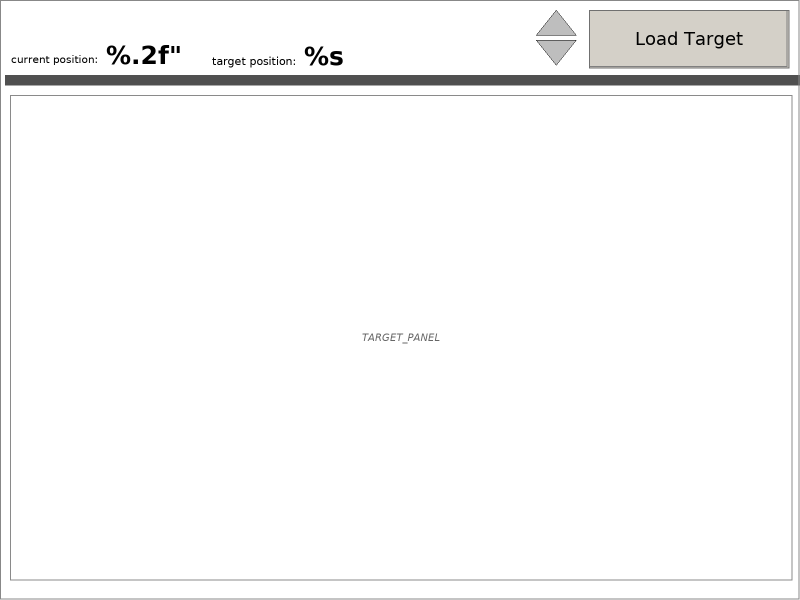
VISUALIZATION MAIN_DASHBOARD  // 800x600
    Rectangle (0,0 810x600)
    Button (589,10 200x58), "Unload Target", colour toggle: GV_HMI.colortoggle[6]
        tap GV_HMI.colortoggle[6]
        OnMouseDown: execute { HMI.bTgtLoaded := FALSE; GV_LIFT.MTS_ALLOWED := FALSE; }
    Rectangle (5,75 795x10)
    Rectangle (12,50 89x19), "current position:"
    Rectangle (103,40 135x30), "%.2f"", text variable: GV_LIFT.CURRENT_POSITION
    Rectangle (208,52 91x19), "target position:"
    Rectangle (301,39 132x34), "%s", text variable: HMI.DisplayTgtPos, invisible if: GV_LIFT.MTS_ALLOWED<>1
    Button (589,10 200x58), "Load Target", colour toggle: GV_HMI.colortoggle[6], invisible if: HMI.bUnload <> 0, input disabled if: HMI.bLoadOK<>1
        tap GV_HMI.colortoggle[6]
        OnMouseDown: execute {
            GV_LIFT.TARGET_POSITION := XML.savedvalues.savedpos[GV_HMI.RowSelect].target;
            GV_HMI.RowSelected := GV_HMI.RowSelect;
            HMI.bTgtLoaded := TRUE;
            GV_LIFT.MTS_ALLOWED := TRUE;
            GV_LIFT.JUST_RAN := FALSE;
        }
    TabControl (10,95 782x485)
        shows TARGET_PANEL()
        shows SAFETY_PANEL()
        shows Visualization_2()
        shows Visualization_2()
        shows Visualization_2()
        [0]: TabTitle=Target Positions
        [1]: TabTitle=Safety Status Panel
    Polygon (536,35) (556,10) (576,35) (576,35) (536,35), colour variable: HMI_Up_Arrow_Indicator.dwUpArrow
    Polygon (536,40) (556,65) (576,40) (576,40) (536,40), colour variable: HMI_Down_Arrow_Indicator.dwDownArrow
END_VISUALIZATION

// ---- VISUs/SAFETY_PANEL.TcVIS
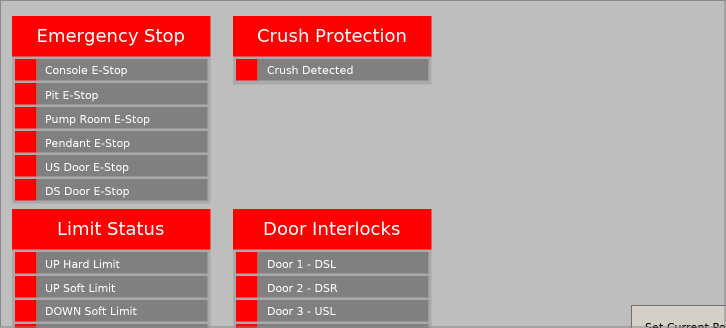
VISUALIZATION SAFETY_PANEL  // 726x328
    Rectangle (233,39 198x45)
    Rectangle (12,38 198x165)
    Rectangle (233,228 198x120)
    Rectangle (12,228 198x144)
    RoundedRectangle (15,276 21x21), colour toggle: HMI.bSoftUpLimFlag
    Rectangle (37,276 170x21)
    Rectangle (42,275 130x27), "UP Soft Limit"
    RoundedRectangle (15,300 21x21), colour toggle: HMI.bSoftDownLimFlag
    Rectangle (37,300 170x21)
    Rectangle (42,298 130x27), "DOWN Soft Limit"
    RoundedRectangle (15,324 21x21), colour variable: HMI_Hard_Limits.DownHardLimit
    Rectangle (37,324 170x21)
    Rectangle (42,322 130x27), "DOWN Hard Limit"
    RoundedRectangle (12,209 198x40), "Limit Status", colour toggle: HMI.bLimitHeaderFlag
    RoundedRectangle (236,252 21x21), colour variable: HMI_Door_Toggle.dwDoor1
    Rectangle (258,252 170x21)
    Rectangle (264,251 130x27), "Door 1 - DSL"
    RoundedRectangle (236,276 21x21), colour variable: HMI_Door_Toggle.dwDoor2
    Rectangle (258,276 170x21)
    Rectangle (264,275 130x27), "Door 2 - DSR"
    RoundedRectangle (236,300 21x21), colour variable: HMI_Door_Toggle.dwDoor3
    Rectangle (258,300 170x21)
    Rectangle (264,298 130x27), "Door 3 - USL"
    RoundedRectangle (236,324 21x21), colour variable: HMI_Door_Toggle.dwDoor4
    Rectangle (258,324 170x21)
    Rectangle (264,322 130x27), "Door 4 - USR"
    RoundedRectangle (233,209 198x40), "Door Interlocks", colour variable: HMI_Door_Toggle.dwDoorFlag
    RoundedRectangle (15,59 21x21), colour toggle: GV_LIFT.CONSOLE_ESTOP_INDICATOR_IN
    Rectangle (37,59 170x21)
    Rectangle (42,57 130x27), "Console E-Stop"
    RoundedRectangle (15,83 21x21), colour toggle: GV_LIFT.PIT_ESTOP_INDICATOR_IN
    Rectangle (37,83 170x21)
    Rectangle (42,82 130x27), "Pit E-Stop"
    RoundedRectangle (15,131 21x21), colour toggle: GV_LIFT.REMOTE_ESTOP_INDICATOR_IN
    Rectangle (37,131 170x21)
    Rectangle (42,130 130x27), "Pendant E-Stop"
    RoundedRectangle (15,155 21x21), colour toggle: GV_LIFT.UPSTAGE_ESTOP_INDICATOR_IN
    Rectangle (37,155 170x21)
    Rectangle (42,154 130x27), "US Door E-Stop"
    RoundedRectangle (12,16 198x40), "Emergency Stop", colour toggle: GV_LIFT.ESTOP_INDICATOR_OUT
    RoundedRectangle (15,179 21x21), colour toggle: GV_LIFT.DOWNSTAGE_ESTOP_INDICATOR_IN
    Rectangle (37,179 170x21)
    Rectangle (42,178 130x27), "DS Door E-Stop"
    RoundedRectangle (236,59 21x21), colour variable: HMI_Crush_Indicator.dwCrushFlag
    Rectangle (258,59 170x21)
    Rectangle (264,57 130x27), "Crush Detected"
    RoundedRectangle (233,16 198x40), "Crush Protection", colour variable: HMI_Crush_Indicator.dwCrushFlag
    Button (631,305 138x45), "Set Current Position", colour toggle: (GV_HMI.colortoggle[1])<>0
        tap GV_HMI.colortoggle[1]
        OnDialogClosed: execute { MOVE_TO_POSITION.bRecalculatePosition := TRUE; }
        OnMouseDown: write GV_HMI.updatedPos via VisuDialogs.Numpad, title 'Current Position'
    Button (631,355 138x45), "Set UP Soft Limit", colour toggle: (GV_HMI.colortoggle[2])<>0
        tap GV_HMI.colortoggle[2]
        OnMouseDown: write XML.savedvalues.UpSoftLim via VisuDialogs.Numpad, title 'Up Soft Limit'
    Button (631,405 138x45), "Set DOWN Soft Limit", colour toggle: (GV_HMI.colortoggle[3])<>0
        tap GV_HMI.colortoggle[3]
        OnMouseDown: write XML.savedvalues.DownSoftLim via VisuDialogs.Numpad, title 'Down Soft Limit'
    RoundedRectangle (15,348 21x21), colour variable: HMI_Ultimate_Limit.DownUltLimit
    Rectangle (37,348 170x21)
    Rectangle (42,346 130x27), "DOWN Ultimate Limit"
    RoundedRectangle (15,252 21x21), colour variable: HMI_Hard_Limits.UpHardLimit
    Rectangle (37,252 170x21)
    Rectangle (42,251 130x27), "UP Hard Limit"
    Rectangle (472,362 140x30), "UP Soft Limit %.2f"", text variable: XML.savedvalues.UpSoftLim
    Rectangle (472,412 140x30), "DOWN Soft Limit: %.2f"", text variable: XML.savedvalues.DownSoftLim
    RoundedRectangle (15,107 21x21), colour toggle: GV_LIFT.PUMP_ESTOP_INDICATOR_IN
    Rectangle (37,107 170x21)
    Rectangle (42,106 130x27), "Pump Room E-Stop"
END_VISUALIZATION

// ---- VISUs/TARGET_PANEL.TcVIS
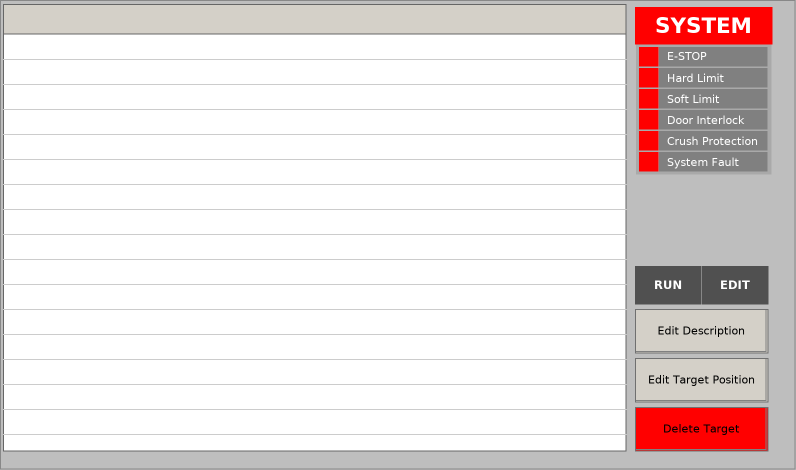
VISUALIZATION TARGET_PANEL  // 796x470
    Button (635,358 133x44), "Edit Target Position", colour toggle: (GV_HMI.ColorToggle[2])<>0, invisible if: HMI.bEditEnable<>1
        tap GV_HMI.ColorToggle[2]
        OnDialogClosed: execute {
            IF XML.savedvalues.savedpos[GV_HMI.RowSelect].target <= XML.savedvalues.UpSoftLim AND XML.savedvalues.savedpos[GV_HMI.RowSelect].target >= XML.savedvalues.DownSoftLim THEN
            	XML.savedvalues.savedpos[GV_HMI.RowSelect].targetclear := TRUE;
            ELSE
            	XML.savedvalues.savedpos[GV_HMI.RowSelect].targetclear := FALSE;
            END_IF
        }
        OnMouseDown: write XML.savedvalues.savedpos[.GV_HMI.RowSelect].target via VisuDialogs.Numpad, min XML.savedvalues.DownSoftLim, max XML.savedvalues.UpSoftLim, title 'Target Position'
    Button (635,309 133x44), "Edit Description", colour toggle: GV_HMI.ColorToggle[3], invisible if: HMI.bEditEnable<>1
        tap GV_HMI.ColorToggle[3]
        OnMouseDown: write XML.savedvalues.savedpos[.GV_HMI.RowSelect].description via VisuDialogs.Keypad, title 'Edit Target Description'
        OnMouseDown: execute {
            IF XML.savedvalues.savedpos[GV_HMI.RowSelect].target <= XML.savedvalues.UpSoftLim AND XML.savedvalues.savedpos[GV_HMI.RowSelect].target >= XML.savedvalues.DownSoftLim THEN
            	XML.savedvalues.savedpos[GV_HMI.RowSelect].targetclear := TRUE;
            ELSE
            	XML.savedvalues.savedpos[GV_HMI.RowSelect].targetclear := FALSE;
            END_IF
        }
    Table (3,4 623x447), data array: HMI.displayvalues
        p1420305297: GV_HMI.ColumnSelect
        p1137915858: GV_HMI.RowSelect
        p3854506369: HMI.displayvalues[INDEX].target
        p1892666644: HMI.displayvalues[INDEX].description
        p2232123230: Target Position
        p511219082: Description
    Rectangle (636,27 135x147)
    RoundedRectangle (639,47 19x19), colour toggle: GV_LIFT.ESTOP_INDICATOR_OUT
    RoundedRectangle (639,68 19x19), colour variable: HMI_Hard_Limits.HardLimitFlag
    RoundedRectangle (639,89 19x19), colour toggle: HMI.bSoftLimFlag
    RoundedRectangle (639,110 19x19), colour variable: HMI_Door_Toggle.dwDoorFlag
    RoundedRectangle (635,7 137x37), "SYSTEM", colour toggle: HMI_System_Indicator.bSystemFlag
    RoundedRectangle (639,131 19x19), colour variable: HMI_Crush_Indicator.dwCrushFlag
    RoundedRectangle (639,152 19x19), colour toggle: GV_LIFT.SYSTEM_FAULT <>1
    Rectangle (659,47 108x19)
    Rectangle (664,44 100x25), "E-STOP"
    Rectangle (659,68 108x19)
    Rectangle (664,66 100x25), "Hard Limit"
    Rectangle (659,89 108x19)
    Rectangle (664,87 100x25), "Soft Limit"
    Rectangle (659,110 108x19)
    Rectangle (664,108 100x25), "Door Interlock"
    Rectangle (659,131 108x19)
    Rectangle (664,129 100x25), "Crush Protection"
    Rectangle (659,152 108x19)
    Rectangle (664,150 100x25), "System Fault"
    Button (635,407 133x44), "Delete Target", colour toggle: (GV_HMI.ColorToggle[1])<>0, invisible if: HMI.bEditEnable<>1
        tap GV_HMI.ColorToggle[1]
        OnMouseDown: execute {
            XML.savedvalues.savedpos[GV_HMI.RowSelect].targetclear := FALSE;
            XML.savedvalues.savedpos[GV_HMI.RowSelect].target := 0.00;
            XML.savedvalues.savedpos[GV_HMI.RowSelect].description := '';
        }
    Rectangle (635,266 66x38), "RUN", colour toggle: HMI.bEditEnable<>0
        OnMouseDown: execute { HMI.bEditEnable:=FALSE; }
    Rectangle (702,266 66x38), "EDIT", colour toggle: HMI.bEditEnable<>1
        OnMouseDown: execute { HMI.bEditEnable:=TRUE; }
END_VISUALIZATION
